ABB RAPID module: P903.mod

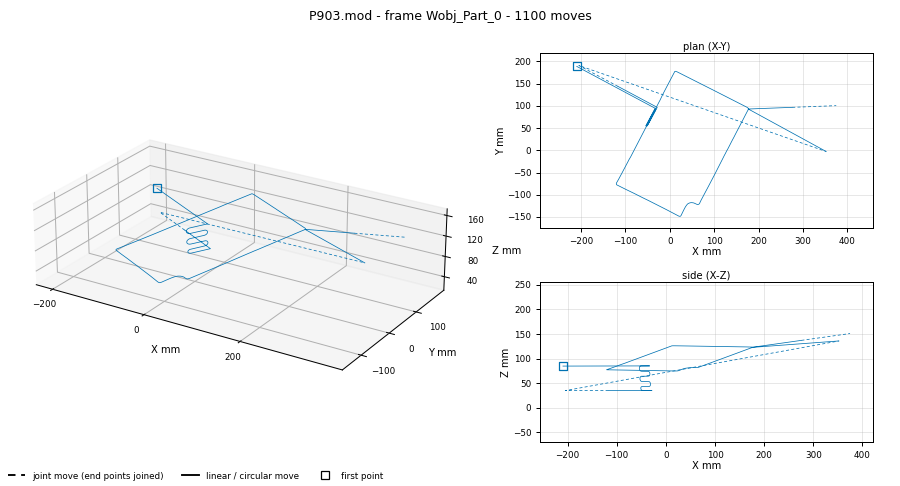
[picture p0: tool path of P903.mod in frame Wobj_Part_0, 1100 of 1110 moves have a stored position in this frame; points joined in program order, loops and branches not executed]
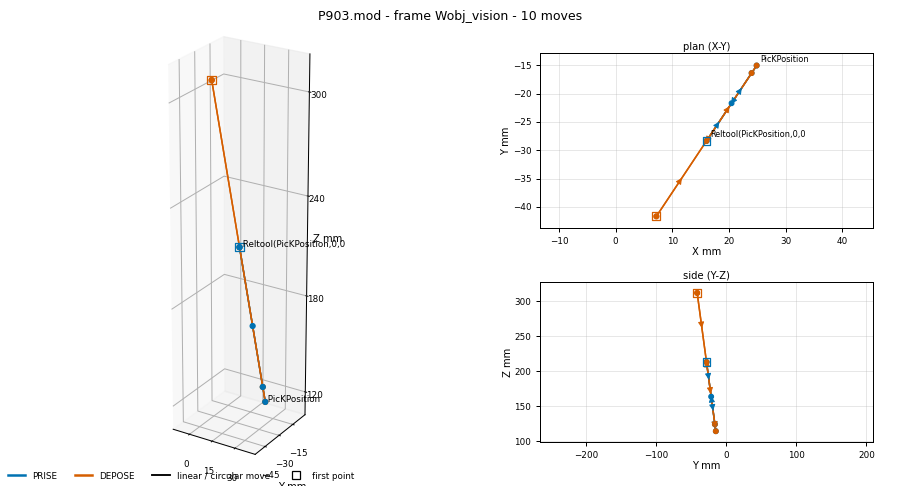
[picture p1: tool path of P903.mod in frame Wobj_vision, 10 of 1110 moves have a stored position in this frame; points joined in program order, loops and branches not executed]
MODULE P903

    ! Nom         :P903
    ! Description :
    ! Créé le     :01/06/2023 15:01:56

    LOCAL CONST SPEEDDATA VitesseLente :=[10,500,0,0];
	LOCAL CONST SPEEDDATA VitesseRapide :=[30,500,0,0];
	LOCAL CONST SPEEDDATA VitesseTronconnage :=[2,500,0,0];
	LOCAL CONST SPEEDDATA VitesseTronconnageApp :=[10,500,0,0];
    !
    !Point de prise
    LOCAL PERS Robtarget PicKPosition := [[24.8984358330106,-15.047813549993,114.680940912607],[0.072391542701378,-0.511697076202154,0.855414280882458,0.0345249882523983],[0,0,0,0],[8.999999E+09,8.999999E+09,8.999999E+09,8.999999E+09,8.999999E+09,8.999999E+09]];
	LOCAL PERS Pose Ref := [[0,0,0],[1,0,0,0]];
    !
    !Declaration des points de meulage

    !Tr_meulage_motif_1 : Meulage d'un motif
    LOCAL CONST Robtarget Tr_meulage_motif_1_0 := [[-32.91730859375,94.6825546875,85.178703125],[0.363951430919515,-0.363241574410581,0.605870778174484,-0.607054787235555],[0,0,0,0],[8.999999E+09,8.999999E+09,8.999999E+09,8.999999E+09,8.999999E+09,8.999999E+09]];
    LOCAL CONST Robtarget Tr_meulage_motif_1_1 := [[-33.3889453125,93.8007578125,85.178671875],[0.363951430919515,-0.363241574410581,0.605870778174484,-0.607054787235555],[0,0,0,0],[8.999999E+09,8.999999E+09,8.999999E+09,8.999999E+09,8.999999E+09,8.999999E+09]];
    LOCAL CONST Robtarget Tr_meulage_motif_1_2 := [[-33.8605859375,92.91896875,85.1786484375],[0.363951430919515,-0.363241574410581,0.605870778174484,-0.607054787235555],[0,0,0,0],[8.999999E+09,8.999999E+09,8.999999E+09,8.999999E+09,8.999999E+09,8.999999E+09]];
    LOCAL CONST Robtarget Tr_meulage_motif_1_3 := [[-34.33222265625,92.037171875,85.178625],[0.363951430919515,-0.363241574410581,0.605870778174484,-0.607054787235555],[0,0,0,0],[8.999999E+09,8.999999E+09,8.999999E+09,8.999999E+09,8.999999E+09,8.999999E+09]];
    LOCAL CONST Robtarget Tr_meulage_motif_1_4 := [[-34.803859375,91.1553828125,85.1786015625],[0.363951430919515,-0.363241574410581,0.605870778174484,-0.607054787235555],[0,0,0,0],[8.999999E+09,8.999999E+09,8.999999E+09,8.999999E+09,8.999999E+09,8.999999E+09]];
    LOCAL CONST Robtarget Tr_meulage_motif_1_5 := [[-35.27549609375,90.2735859375,85.178578125],[0.363951430919515,-0.363241574410581,0.605870778174484,-0.607054787235555],[0,0,0,0],[8.999999E+09,8.999999E+09,8.999999E+09,8.999999E+09,8.999999E+09,8.999999E+09]];
    LOCAL CONST Robtarget Tr_meulage_motif_1_6 := [[-35.74713671875,89.391796875,85.178546875],[0.363951430919515,-0.363241574410581,0.605870778174484,-0.607054787235555],[0,0,0,0],[8.999999E+09,8.999999E+09,8.999999E+09,8.999999E+09,8.999999E+09,8.999999E+09]];
    LOCAL CONST Robtarget Tr_meulage_motif_1_7 := [[-36.2187734375,88.5100078125,85.1785234375],[0.363951430919515,-0.363241574410581,0.605870778174484,-0.607054787235555],[0,0,0,0],[8.999999E+09,8.999999E+09,8.999999E+09,8.999999E+09,8.999999E+09,8.999999E+09]];
    LOCAL CONST Robtarget Tr_meulage_motif_1_8 := [[-36.69041015625,87.6282109375,85.1785],[0.363951430919515,-0.363241574410581,0.605870778174484,-0.607054787235555],[0,0,0,0],[8.999999E+09,8.999999E+09,8.999999E+09,8.999999E+09,8.999999E+09,8.999999E+09]];
    LOCAL CONST Robtarget Tr_meulage_motif_1_9 := [[-37.162046875,86.746421875,85.1784765625],[0.363951430919515,-0.363241574410581,0.605870778174484,-0.607054787235555],[0,0,0,0],[8.999999E+09,8.999999E+09,8.999999E+09,8.999999E+09,8.999999E+09,8.999999E+09]];
    LOCAL CONST Robtarget Tr_meulage_motif_1_10 := [[-37.6336875,85.864625,85.1784453125],[0.363951430919515,-0.363241574410581,0.605870778174484,-0.607054787235555],[0,0,0,0],[8.999999E+09,8.999999E+09,8.999999E+09,8.999999E+09,8.999999E+09,8.999999E+09]];
    LOCAL CONST Robtarget Tr_meulage_motif_1_11 := [[-38.10532421875,84.9828359375,85.178421875],[0.363951430919515,-0.363241574410581,0.605870778174484,-0.607054787235555],[0,0,0,0],[8.999999E+09,8.999999E+09,8.999999E+09,8.999999E+09,8.999999E+09,8.999999E+09]];
    LOCAL CONST Robtarget Tr_meulage_motif_1_12 := [[-38.5769609375,84.1010390625,85.1783984375],[0.363951430919515,-0.363241574410581,0.605870778174484,-0.607054787235555],[0,0,0,0],[8.999999E+09,8.999999E+09,8.999999E+09,8.999999E+09,8.999999E+09,8.999999E+09]];
    LOCAL CONST Robtarget Tr_meulage_motif_1_13 := [[-39.04859765625,83.21925,85.178375],[0.363951430919515,-0.363241574410581,0.605870778174484,-0.607054787235555],[0,0,0,0],[8.999999E+09,8.999999E+09,8.999999E+09,8.999999E+09,8.999999E+09,8.999999E+09]];
    LOCAL CONST Robtarget Tr_meulage_motif_1_14 := [[-39.52023828125,82.3374609375,85.1783515625],[0.363951430919515,-0.363241574410581,0.605870778174484,-0.607054787235555],[0,0,0,0],[8.999999E+09,8.999999E+09,8.999999E+09,8.999999E+09,8.999999E+09,8.999999E+09]];
    LOCAL CONST Robtarget Tr_meulage_motif_1_15 := [[-39.991875,81.4556640625,85.1783203125],[0.363951430919515,-0.363241574410581,0.605870778174484,-0.607054787235555],[0,0,0,0],[8.999999E+09,8.999999E+09,8.999999E+09,8.999999E+09,8.999999E+09,8.999999E+09]];
    LOCAL CONST Robtarget Tr_meulage_motif_1_16 := [[-40.46351171875,80.573875,85.178296875],[0.363951430919515,-0.363241574410581,0.605870778174484,-0.607054787235555],[0,0,0,0],[8.999999E+09,8.999999E+09,8.999999E+09,8.999999E+09,8.999999E+09,8.999999E+09]];
    LOCAL CONST Robtarget Tr_meulage_motif_1_17 := [[-40.9351484375,79.692078125,85.1782734375],[0.363951430919515,-0.363241574410581,0.605870778174484,-0.607054787235555],[0,0,0,0],[8.999999E+09,8.999999E+09,8.999999E+09,8.999999E+09,8.999999E+09,8.999999E+09]];
    LOCAL CONST Robtarget Tr_meulage_motif_1_18 := [[-41.4067890625,78.8102890625,85.17825],[0.363951430919515,-0.363241574410581,0.605870778174484,-0.607054787235555],[0,0,0,0],[8.999999E+09,8.999999E+09,8.999999E+09,8.999999E+09,8.999999E+09,8.999999E+09]];
    LOCAL CONST Robtarget Tr_meulage_motif_1_19 := [[-41.87842578125,77.9284921875,85.1782265625],[0.363951430919515,-0.363241574410581,0.605870778174484,-0.607054787235555],[0,0,0,0],[8.999999E+09,8.999999E+09,8.999999E+09,8.999999E+09,8.999999E+09,8.999999E+09]];
    LOCAL CONST Robtarget Tr_meulage_motif_1_20 := [[-42.3500625,77.046703125,85.1781953125],[0.363951430919515,-0.363241574410581,0.605870778174484,-0.607054787235555],[0,0,0,0],[8.999999E+09,8.999999E+09,8.999999E+09,8.999999E+09,8.999999E+09,8.999999E+09]];
    LOCAL CONST Robtarget Tr_meulage_motif_1_21 := [[-42.82169921875,76.1649140625,85.178171875],[0.363951430919515,-0.363241574410581,0.605870778174484,-0.607054787235555],[0,0,0,0],[8.999999E+09,8.999999E+09,8.999999E+09,8.999999E+09,8.999999E+09,8.999999E+09]];
    LOCAL CONST Robtarget Tr_meulage_motif_1_22 := [[-43.29333984375,75.2831171875,85.1781484375],[0.363951430919515,-0.363241574410581,0.605870778174484,-0.607054787235555],[0,0,0,0],[8.999999E+09,8.999999E+09,8.999999E+09,8.999999E+09,8.999999E+09,8.999999E+09]];
    LOCAL CONST Robtarget Tr_meulage_motif_1_23 := [[-43.7649765625,74.401328125,85.178125],[0.363951430919515,-0.363241574410581,0.605870778174484,-0.607054787235555],[0,0,0,0],[8.999999E+09,8.999999E+09,8.999999E+09,8.999999E+09,8.999999E+09,8.999999E+09]];
    LOCAL CONST Robtarget Tr_meulage_motif_1_24 := [[-44.23661328125,73.51953125,85.17809375],[0.363951430919515,-0.363241574410581,0.605870778174484,-0.607054787235555],[0,0,0,0],[8.999999E+09,8.999999E+09,8.999999E+09,8.999999E+09,8.999999E+09,8.999999E+09]];
    LOCAL CONST Robtarget Tr_meulage_motif_1_25 := [[-44.70825,72.6377421875,85.1780703125],[0.363951430919515,-0.363241574410581,0.605870778174484,-0.607054787235555],[0,0,0,0],[8.999999E+09,8.999999E+09,8.999999E+09,8.999999E+09,8.999999E+09,8.999999E+09]];
    LOCAL CONST Robtarget Tr_meulage_motif_1_26 := [[-45.179890625,71.7559453125,85.178046875],[0.363951430919515,-0.363241574410581,0.605870778174484,-0.607054787235555],[0,0,0,0],[8.999999E+09,8.999999E+09,8.999999E+09,8.999999E+09,8.999999E+09,8.999999E+09]];
    LOCAL CONST Robtarget Tr_meulage_motif_1_27 := [[-45.65152734375,70.87415625,85.1780234375],[0.363951430919515,-0.363241574410581,0.605870778174484,-0.607054787235555],[0,0,0,0],[8.999999E+09,8.999999E+09,8.999999E+09,8.999999E+09,8.999999E+09,8.999999E+09]];
    LOCAL CONST Robtarget Tr_meulage_motif_1_28 := [[-46.1231640625,69.9923671875,85.178],[0.363951430919515,-0.363241574410581,0.605870778174484,-0.607054787235555],[0,0,0,0],[8.999999E+09,8.999999E+09,8.999999E+09,8.999999E+09,8.999999E+09,8.999999E+09]];
    LOCAL CONST Robtarget Tr_meulage_motif_1_29 := [[-46.59480078125,69.1105703125,85.17796875],[0.363951430919515,-0.363241574410581,0.605870778174484,-0.607054787235555],[0,0,0,0],[8.999999E+09,8.999999E+09,8.999999E+09,8.999999E+09,8.999999E+09,8.999999E+09]];
    LOCAL CONST Robtarget Tr_meulage_motif_1_30 := [[-47.06644140625,68.22878125,85.1779453125],[0.363951430919515,-0.363241574410581,0.605870778174484,-0.607054787235555],[0,0,0,0],[8.999999E+09,8.999999E+09,8.999999E+09,8.999999E+09,8.999999E+09,8.999999E+09]];
    LOCAL CONST Robtarget Tr_meulage_motif_1_31 := [[-47.538078125,67.346984375,85.177921875],[0.363951430919515,-0.363241574410581,0.605870778174484,-0.607054787235555],[0,0,0,0],[8.999999E+09,8.999999E+09,8.999999E+09,8.999999E+09,8.999999E+09,8.999999E+09]];
    LOCAL CONST Robtarget Tr_meulage_motif_1_32 := [[-48.00971484375,66.4651953125,85.1778984375],[0.363951430919515,-0.363241574410581,0.605870778174484,-0.607054787235555],[0,0,0,0],[8.999999E+09,8.999999E+09,8.999999E+09,8.999999E+09,8.999999E+09,8.999999E+09]];
    LOCAL CONST Robtarget Tr_meulage_motif_1_33 := [[-48.4813515625,65.5833984375,85.1778671875],[0.363951430919515,-0.363241574410581,0.605870778174484,-0.607054787235555],[0,0,0,0],[8.999999E+09,8.999999E+09,8.999999E+09,8.999999E+09,8.999999E+09,8.999999E+09]];
    LOCAL CONST Robtarget Tr_meulage_motif_1_34 := [[-48.9529921875,64.701609375,85.17784375],[0.363951430919515,-0.363241574410581,0.605870778174484,-0.607054787235555],[0,0,0,0],[8.999999E+09,8.999999E+09,8.999999E+09,8.999999E+09,8.999999E+09,8.999999E+09]];
    LOCAL CONST Robtarget Tr_meulage_motif_1_35 := [[-49.42462890625,63.81981640625,85.1778203125],[0.363951430919515,-0.363241574410581,0.605870778174484,-0.607054787235555],[0,0,0,0],[8.999999E+09,8.999999E+09,8.999999E+09,8.999999E+09,8.999999E+09,8.999999E+09]];
    LOCAL CONST Robtarget Tr_meulage_motif_1_36 := [[-49.896265625,62.9380234375,85.177796875],[0.363951430919515,-0.363241574410581,0.605870778174484,-0.607054787235555],[0,0,0,0],[8.999999E+09,8.999999E+09,8.999999E+09,8.999999E+09,8.999999E+09,8.999999E+09]];
    LOCAL CONST Robtarget Tr_meulage_motif_1_37 := [[-50.36790234375,62.05623046875,85.1777734375],[0.363951430919515,-0.363241574410581,0.605870778174484,-0.607054787235555],[0,0,0,0],[8.999999E+09,8.999999E+09,8.999999E+09,8.999999E+09,8.999999E+09,8.999999E+09]];
    LOCAL CONST Robtarget Tr_meulage_motif_1_38 := [[-50.83954296875,61.1744375,85.1777421875],[0.363951430919515,-0.363241574410581,0.605870778174484,-0.607054787235555],[0,0,0,0],[8.999999E+09,8.999999E+09,8.999999E+09,8.999999E+09,8.999999E+09,8.999999E+09]];
    LOCAL CONST Robtarget Tr_meulage_motif_1_39 := [[-51.3013984375,60.2958515625,85.067359375],[0.363951430919515,-0.363241574410581,0.605870778174484,-0.607054787235555],[0,0,0,0],[8.999999E+09,8.999999E+09,8.999999E+09,8.999999E+09,8.999999E+09,8.999999E+09]];
    LOCAL CONST Robtarget Tr_meulage_motif_1_40 := [[-51.7358203125,59.45483203125,84.856578125],[0.363951430919515,-0.363241574410581,0.605870778174484,-0.607054787235555],[0,0,0,0],[8.999999E+09,8.999999E+09,8.999999E+09,8.999999E+09,8.999999E+09,8.999999E+09]];
    LOCAL CONST Robtarget Tr_meulage_motif_1_41 := [[-52.12257421875,58.694671875,84.58528125],[0.363951430919515,-0.363241574410581,0.605870778174484,-0.607054787235555],[0,0,0,0],[8.999999E+09,8.999999E+09,8.999999E+09,8.999999E+09,8.999999E+09,8.999999E+09]];
    LOCAL CONST Robtarget Tr_meulage_motif_1_42 := [[-52.4606171875,58.025015625,84.3098984375],[0.363951430919515,-0.363241574410581,0.605870778174484,-0.607054787235555],[0,0,0,0],[8.999999E+09,8.999999E+09,8.999999E+09,8.999999E+09,8.999999E+09,8.999999E+09]];
    LOCAL CONST Robtarget Tr_meulage_motif_1_43 := [[-52.94496484375,57.0354296875,83.695015625],[0.363951430919515,-0.363241574410581,0.605870778174484,-0.607054787235555],[0,0,0,0],[8.999999E+09,8.999999E+09,8.999999E+09,8.999999E+09,8.999999E+09,8.999999E+09]];
    LOCAL CONST Robtarget Tr_meulage_motif_1_44 := [[-53.37976953125,56.10688671875,82.84909375],[0.363951430919515,-0.363241574410581,0.605870778174484,-0.607054787235555],[0,0,0,0],[8.999999E+09,8.999999E+09,8.999999E+09,8.999999E+09,8.999999E+09,8.999999E+09]];
    LOCAL CONST Robtarget Tr_meulage_motif_1_45 := [[-53.72146875,55.328390625,81.8273125],[0.363951430919515,-0.363241574410581,0.605870778174484,-0.607054787235555],[0,0,0,0],[8.999999E+09,8.999999E+09,8.999999E+09,8.999999E+09,8.999999E+09,8.999999E+09]];
    LOCAL CONST Robtarget Tr_meulage_motif_1_46 := [[-53.888375,54.86409765625,80.7134296875],[0.363951430919515,-0.363241574410581,0.605870778174484,-0.607054787235555],[0,0,0,0],[8.999999E+09,8.999999E+09,8.999999E+09,8.999999E+09,8.999999E+09,8.999999E+09]];
    LOCAL CONST Robtarget Tr_meulage_motif_1_47 := [[-53.86165625,54.81913671875,80.0188984375],[0.363951430919515,-0.363241574410581,0.605870778174484,-0.607054787235555],[0,0,0,0],[8.999999E+09,8.999999E+09,8.999999E+09,8.999999E+09,8.999999E+09,8.999999E+09]];
    LOCAL CONST Robtarget Tr_meulage_motif_1_48 := [[-53.824140625,54.79908984375,79.359015625],[0.363951430919515,-0.363241574410581,0.605870778174484,-0.607054787235555],[0,0,0,0],[8.999999E+09,8.999999E+09,8.999999E+09,8.999999E+09,8.999999E+09,8.999999E+09]];
    LOCAL CONST Robtarget Tr_meulage_motif_1_49 := [[-53.76075390625,54.82743359375,78.699296875],[0.363951430919515,-0.363241574410581,0.605870778174484,-0.607054787235555],[0,0,0,0],[8.999999E+09,8.999999E+09,8.999999E+09,8.999999E+09,8.999999E+09,8.999999E+09]];
    LOCAL CONST Robtarget Tr_meulage_motif_1_50 := [[-53.463265625,55.233359375,77.59984375],[0.363951430919515,-0.363241574410581,0.605870778174484,-0.607054787235555],[0,0,0,0],[8.999999E+09,8.999999E+09,8.999999E+09,8.999999E+09,8.999999E+09,8.999999E+09]];
    LOCAL CONST Robtarget Tr_meulage_motif_1_51 := [[-53.002140625,55.95820703125,76.5953203125],[0.363951430919515,-0.363241574410581,0.605870778174484,-0.607054787235555],[0,0,0,0],[8.999999E+09,8.999999E+09,8.999999E+09,8.999999E+09,8.999999E+09,8.999999E+09]];
    LOCAL CONST Robtarget Tr_meulage_motif_1_52 := [[-52.4724375,56.83551171875,75.7681875],[0.363951430919515,-0.363241574410581,0.605870778174484,-0.607054787235555],[0,0,0,0],[8.999999E+09,8.999999E+09,8.999999E+09,8.999999E+09,8.999999E+09,8.999999E+09]];
    LOCAL CONST Robtarget Tr_meulage_motif_1_53 := [[-52.12592578125,57.42938671875,75.3732734375],[0.363951430919515,-0.363241574410581,0.605870778174484,-0.607054787235555],[0,0,0,0],[8.999999E+09,8.999999E+09,8.999999E+09,8.999999E+09,8.999999E+09,8.999999E+09]];
    LOCAL CONST Robtarget Tr_meulage_motif_1_54 := [[-51.55203515625,58.435859375,74.88678125],[0.363951430919515,-0.363241574410581,0.605870778174484,-0.607054787235555],[0,0,0,0],[8.999999E+09,8.999999E+09,8.999999E+09,8.999999E+09,8.999999E+09,8.999999E+09]];
    LOCAL CONST Robtarget Tr_meulage_motif_1_55 := [[-51.13850390625,59.17299609375,74.6232578125],[0.363951430919515,-0.363241574410581,0.605870778174484,-0.607054787235555],[0,0,0,0],[8.999999E+09,8.999999E+09,8.999999E+09,8.999999E+09,8.999999E+09,8.999999E+09]];
    LOCAL CONST Robtarget Tr_meulage_motif_1_56 := [[-50.68733984375,59.98862890625,74.419234375],[0.363951430919515,-0.363241574410581,0.605870778174484,-0.607054787235555],[0,0,0,0],[8.999999E+09,8.999999E+09,8.999999E+09,8.999999E+09,8.999999E+09,8.999999E+09]];
    LOCAL CONST Robtarget Tr_meulage_motif_1_57 := [[-50.218234375,60.85087109375,74.310890625],[0.363951430919515,-0.363241574410581,0.605870778174484,-0.607054787235555],[0,0,0,0],[8.999999E+09,8.999999E+09,8.999999E+09,8.999999E+09,8.999999E+09,8.999999E+09]];
    LOCAL CONST Robtarget Tr_meulage_motif_1_58 := [[-49.74383203125,61.72275,74.2005546875],[0.363951430919515,-0.363241574410581,0.605870778174484,-0.607054787235555],[0,0,0,0],[8.999999E+09,8.999999E+09,8.999999E+09,8.999999E+09,8.999999E+09,8.999999E+09]];
    LOCAL CONST Robtarget Tr_meulage_motif_1_59 := [[-49.2721953125,62.60454296875,74.200578125],[0.363951430919515,-0.363241574410581,0.605870778174484,-0.607054787235555],[0,0,0,0],[8.999999E+09,8.999999E+09,8.999999E+09,8.999999E+09,8.999999E+09,8.999999E+09]];
    LOCAL CONST Robtarget Tr_meulage_motif_1_60 := [[-48.8005546875,63.4863359375,74.2006015625],[0.363951430919515,-0.363241574410581,0.605870778174484,-0.607054787235555],[0,0,0,0],[8.999999E+09,8.999999E+09,8.999999E+09,8.999999E+09,8.999999E+09,8.999999E+09]];
    LOCAL CONST Robtarget Tr_meulage_motif_1_61 := [[-48.32891796875,64.36812890625,74.200625],[0.363951430919515,-0.363241574410581,0.605870778174484,-0.607054787235555],[0,0,0,0],[8.999999E+09,8.999999E+09,8.999999E+09,8.999999E+09,8.999999E+09,8.999999E+09]];
    LOCAL CONST Robtarget Tr_meulage_motif_1_62 := [[-47.85728125,65.249921875,74.20065625],[0.363951430919515,-0.363241574410581,0.605870778174484,-0.607054787235555],[0,0,0,0],[8.999999E+09,8.999999E+09,8.999999E+09,8.999999E+09,8.999999E+09,8.999999E+09]];
    LOCAL CONST Robtarget Tr_meulage_motif_1_63 := [[-47.38564453125,66.1317109375,74.2006796875],[0.363951430919515,-0.363241574410581,0.605870778174484,-0.607054787235555],[0,0,0,0],[8.999999E+09,8.999999E+09,8.999999E+09,8.999999E+09,8.999999E+09,8.999999E+09]];
    LOCAL CONST Robtarget Tr_meulage_motif_1_64 := [[-46.91400390625,67.0135078125,74.200703125],[0.363951430919515,-0.363241574410581,0.605870778174484,-0.607054787235555],[0,0,0,0],[8.999999E+09,8.999999E+09,8.999999E+09,8.999999E+09,8.999999E+09,8.999999E+09]];
    LOCAL CONST Robtarget Tr_meulage_motif_1_65 := [[-46.4423671875,67.895296875,74.2007265625],[0.363951430919515,-0.363241574410581,0.605870778174484,-0.607054787235555],[0,0,0,0],[8.999999E+09,8.999999E+09,8.999999E+09,8.999999E+09,8.999999E+09,8.999999E+09]];
    LOCAL CONST Robtarget Tr_meulage_motif_1_66 := [[-45.97073046875,68.77709375,74.20075],[0.363951430919515,-0.363241574410581,0.605870778174484,-0.607054787235555],[0,0,0,0],[8.999999E+09,8.999999E+09,8.999999E+09,8.999999E+09,8.999999E+09,8.999999E+09]];
    LOCAL CONST Robtarget Tr_meulage_motif_1_67 := [[-45.49909375,69.6588828125,74.20078125],[0.363951430919515,-0.363241574410581,0.605870778174484,-0.607054787235555],[0,0,0,0],[8.999999E+09,8.999999E+09,8.999999E+09,8.999999E+09,8.999999E+09,8.999999E+09]];
    LOCAL CONST Robtarget Tr_meulage_motif_1_68 := [[-45.027453125,70.540671875,74.2008046875],[0.363951430919515,-0.363241574410581,0.605870778174484,-0.607054787235555],[0,0,0,0],[8.999999E+09,8.999999E+09,8.999999E+09,8.999999E+09,8.999999E+09,8.999999E+09]];
    LOCAL CONST Robtarget Tr_meulage_motif_1_69 := [[-44.55581640625,71.42246875,74.200828125],[0.363951430919515,-0.363241574410581,0.605870778174484,-0.607054787235555],[0,0,0,0],[8.999999E+09,8.999999E+09,8.999999E+09,8.999999E+09,8.999999E+09,8.999999E+09]];
    LOCAL CONST Robtarget Tr_meulage_motif_1_70 := [[-44.0841796875,72.3042578125,74.2008515625],[0.363951430919515,-0.363241574410581,0.605870778174484,-0.607054787235555],[0,0,0,0],[8.999999E+09,8.999999E+09,8.999999E+09,8.999999E+09,8.999999E+09,8.999999E+09]];
    LOCAL CONST Robtarget Tr_meulage_motif_1_71 := [[-43.61254296875,73.1860546875,74.200875],[0.363951430919515,-0.363241574410581,0.605870778174484,-0.607054787235555],[0,0,0,0],[8.999999E+09,8.999999E+09,8.999999E+09,8.999999E+09,8.999999E+09,8.999999E+09]];
    LOCAL CONST Robtarget Tr_meulage_motif_1_72 := [[-43.14090234375,74.06784375,74.20090625],[0.363951430919515,-0.363241574410581,0.605870778174484,-0.607054787235555],[0,0,0,0],[8.999999E+09,8.999999E+09,8.999999E+09,8.999999E+09,8.999999E+09,8.999999E+09]];
    LOCAL CONST Robtarget Tr_meulage_motif_1_73 := [[-42.669265625,74.949640625,74.2009296875],[0.363951430919515,-0.363241574410581,0.605870778174484,-0.607054787235555],[0,0,0,0],[8.999999E+09,8.999999E+09,8.999999E+09,8.999999E+09,8.999999E+09,8.999999E+09]];
    LOCAL CONST Robtarget Tr_meulage_motif_1_74 := [[-42.19762890625,75.8314296875,74.200953125],[0.363951430919515,-0.363241574410581,0.605870778174484,-0.607054787235555],[0,0,0,0],[8.999999E+09,8.999999E+09,8.999999E+09,8.999999E+09,8.999999E+09,8.999999E+09]];
    LOCAL CONST Robtarget Tr_meulage_motif_1_75 := [[-41.7259921875,76.71321875,74.2009765625],[0.363951430919515,-0.363241574410581,0.605870778174484,-0.607054787235555],[0,0,0,0],[8.999999E+09,8.999999E+09,8.999999E+09,8.999999E+09,8.999999E+09,8.999999E+09]];
    LOCAL CONST Robtarget Tr_meulage_motif_1_76 := [[-41.2543515625,77.595015625,74.2010078125],[0.363951430919515,-0.363241574410581,0.605870778174484,-0.607054787235555],[0,0,0,0],[8.999999E+09,8.999999E+09,8.999999E+09,8.999999E+09,8.999999E+09,8.999999E+09]];
    LOCAL CONST Robtarget Tr_meulage_motif_1_77 := [[-40.78271484375,78.4768046875,74.20103125],[0.363951430919515,-0.363241574410581,0.605870778174484,-0.607054787235555],[0,0,0,0],[8.999999E+09,8.999999E+09,8.999999E+09,8.999999E+09,8.999999E+09,8.999999E+09]];
    LOCAL CONST Robtarget Tr_meulage_motif_1_78 := [[-40.311078125,79.3586015625,74.2010546875],[0.363951430919515,-0.363241574410581,0.605870778174484,-0.607054787235555],[0,0,0,0],[8.999999E+09,8.999999E+09,8.999999E+09,8.999999E+09,8.999999E+09,8.999999E+09]];
    LOCAL CONST Robtarget Tr_meulage_motif_1_79 := [[-39.83944140625,80.240390625,74.201078125],[0.363951430919515,-0.363241574410581,0.605870778174484,-0.607054787235555],[0,0,0,0],[8.999999E+09,8.999999E+09,8.999999E+09,8.999999E+09,8.999999E+09,8.999999E+09]];
    LOCAL CONST Robtarget Tr_meulage_motif_1_80 := [[-39.36780078125,81.1221875,74.2011015625],[0.363951430919515,-0.363241574410581,0.605870778174484,-0.607054787235555],[0,0,0,0],[8.999999E+09,8.999999E+09,8.999999E+09,8.999999E+09,8.999999E+09,8.999999E+09]];
    LOCAL CONST Robtarget Tr_meulage_motif_1_81 := [[-38.8961640625,82.0039765625,74.2011328125],[0.363951430919515,-0.363241574410581,0.605870778174484,-0.607054787235555],[0,0,0,0],[8.999999E+09,8.999999E+09,8.999999E+09,8.999999E+09,8.999999E+09,8.999999E+09]];
    LOCAL CONST Robtarget Tr_meulage_motif_1_82 := [[-38.42452734375,82.8857734375,74.20115625],[0.363951430919515,-0.363241574410581,0.605870778174484,-0.607054787235555],[0,0,0,0],[8.999999E+09,8.999999E+09,8.999999E+09,8.999999E+09,8.999999E+09,8.999999E+09]];
    LOCAL CONST Robtarget Tr_meulage_motif_1_83 := [[-37.952890625,83.7675625,74.2011796875],[0.363951430919515,-0.363241574410581,0.605870778174484,-0.607054787235555],[0,0,0,0],[8.999999E+09,8.999999E+09,8.999999E+09,8.999999E+09,8.999999E+09,8.999999E+09]];
    LOCAL CONST Robtarget Tr_meulage_motif_1_84 := [[-37.48125,84.6493515625,74.201203125],[0.363951430919515,-0.363241574410581,0.605870778174484,-0.607054787235555],[0,0,0,0],[8.999999E+09,8.999999E+09,8.999999E+09,8.999999E+09,8.999999E+09,8.999999E+09]];
    LOCAL CONST Robtarget Tr_meulage_motif_1_85 := [[-37.00961328125,85.5311484375,74.2012265625],[0.363951430919515,-0.363241574410581,0.605870778174484,-0.607054787235555],[0,0,0,0],[8.999999E+09,8.999999E+09,8.999999E+09,8.999999E+09,8.999999E+09,8.999999E+09]];
    LOCAL CONST Robtarget Tr_meulage_motif_1_86 := [[-36.5379765625,86.4129375,74.2012578125],[0.363951430919515,-0.363241574410581,0.605870778174484,-0.607054787235555],[0,0,0,0],[8.999999E+09,8.999999E+09,8.999999E+09,8.999999E+09,8.999999E+09,8.999999E+09]];
    LOCAL CONST Robtarget Tr_meulage_motif_1_87 := [[-36.06633984375,87.294734375,74.20128125],[0.363951430919515,-0.363241574410581,0.605870778174484,-0.607054787235555],[0,0,0,0],[8.999999E+09,8.999999E+09,8.999999E+09,8.999999E+09,8.999999E+09,8.999999E+09]];
    LOCAL CONST Robtarget Tr_meulage_motif_1_88 := [[-35.59469921875,88.1765234375,74.2013046875],[0.363951430919515,-0.363241574410581,0.605870778174484,-0.607054787235555],[0,0,0,0],[8.999999E+09,8.999999E+09,8.999999E+09,8.999999E+09,8.999999E+09,8.999999E+09]];
    LOCAL CONST Robtarget Tr_meulage_motif_1_89 := [[-35.120296875,89.04840625,74.09096875],[0.363951430919515,-0.363241574410581,0.605870778174484,-0.607054787235555],[0,0,0,0],[8.999999E+09,8.999999E+09,8.999999E+09,8.999999E+09,8.999999E+09,8.999999E+09]];
    LOCAL CONST Robtarget Tr_meulage_motif_1_90 := [[-34.66191015625,89.8766171875,73.8802421875],[0.363951430919515,-0.363241574410581,0.605870778174484,-0.607054787235555],[0,0,0,0],[8.999999E+09,8.999999E+09,8.999999E+09,8.999999E+09,8.999999E+09,8.999999E+09]];
    LOCAL CONST Robtarget Tr_meulage_motif_1_91 := [[-34.2443125,90.620296875,73.6089765625],[0.363951430919515,-0.363241574410581,0.605870778174484,-0.607054787235555],[0,0,0,0],[8.999999E+09,8.999999E+09,8.999999E+09,8.999999E+09,8.999999E+09,8.999999E+09]];
    LOCAL CONST Robtarget Tr_meulage_motif_1_92 := [[-33.89148828125,91.2384765625,73.30546875],[0.363951430919515,-0.363241574410581,0.605870778174484,-0.607054787235555],[0,0,0,0],[8.999999E+09,8.999999E+09,8.999999E+09,8.999999E+09,8.999999E+09,8.999999E+09]];
    LOCAL CONST Robtarget Tr_meulage_motif_1_93 := [[-33.36600390625,92.130578125,72.6443359375],[0.363951430919515,-0.363241574410581,0.605870778174484,-0.607054787235555],[0,0,0,0],[8.999999E+09,8.999999E+09,8.999999E+09,8.999999E+09,8.999999E+09,8.999999E+09]];
    LOCAL CONST Robtarget Tr_meulage_motif_1_94 := [[-32.8894453125,92.8985546875,71.7442890625],[0.363951430919515,-0.363241574410581,0.605870778174484,-0.607054787235555],[0,0,0,0],[8.999999E+09,8.999999E+09,8.999999E+09,8.999999E+09,8.999999E+09,8.999999E+09]];
    LOCAL CONST Robtarget Tr_meulage_motif_1_95 := [[-32.5777890625,93.3385703125,70.7004375],[0.363951430919515,-0.363241574410581,0.605870778174484,-0.607054787235555],[0,0,0,0],[8.999999E+09,8.999999E+09,8.999999E+09,8.999999E+09,8.999999E+09,8.999999E+09]];
    LOCAL CONST Robtarget Tr_meulage_motif_1_96 := [[-32.451310546875,93.4804921875,70.0086640625],[0.363951430919515,-0.363241574410581,0.605870778174484,-0.607054787235555],[0,0,0,0],[8.999999E+09,8.999999E+09,8.999999E+09,8.999999E+09,8.999999E+09,8.999999E+09]];
    LOCAL CONST Robtarget Tr_meulage_motif_1_97 := [[-32.377513671875,93.5134453125,69.2402578125],[0.363951430919515,-0.363241574410581,0.605870778174484,-0.607054787235555],[0,0,0,0],[8.999999E+09,8.999999E+09,8.999999E+09,8.999999E+09,8.999999E+09,8.999999E+09]];
    LOCAL CONST Robtarget Tr_meulage_motif_1_98 := [[-32.36540625,93.4310859375,68.4719765625],[0.363951430919515,-0.363241574410581,0.605870778174484,-0.607054787235555],[0,0,0,0],[8.999999E+09,8.999999E+09,8.999999E+09,8.999999E+09,8.999999E+09,8.999999E+09]];
    LOCAL CONST Robtarget Tr_meulage_motif_1_99 := [[-32.500427734375,93.0274921875,67.3660078125],[0.363951430919515,-0.363241574410581,0.605870778174484,-0.607054787235555],[0,0,0,0],[8.999999E+09,8.999999E+09,8.999999E+09,8.999999E+09,8.999999E+09,8.999999E+09]];
    LOCAL CONST Robtarget Tr_meulage_motif_1_100 := [[-32.66260546875,92.6443984375,66.7815234375],[0.363951430919515,-0.363241574410581,0.605870778174484,-0.607054787235555],[0,0,0,0],[8.999999E+09,8.999999E+09,8.999999E+09,8.999999E+09,8.999999E+09,8.999999E+09]];
    LOCAL CONST Robtarget Tr_meulage_motif_1_101 := [[-33.03067578125,91.8352421875,65.89621875],[0.363951430919515,-0.363241574410581,0.605870778174484,-0.607054787235555],[0,0,0,0],[8.999999E+09,8.999999E+09,8.999999E+09,8.999999E+09,8.999999E+09,8.999999E+09]];
    LOCAL CONST Robtarget Tr_meulage_motif_1_102 := [[-33.28340234375,91.3062265625,65.48274609375],[0.363951430919515,-0.363241574410581,0.605870778174484,-0.607054787235555],[0,0,0,0],[8.999999E+09,8.999999E+09,8.999999E+09,8.999999E+09,8.999999E+09,8.999999E+09]];
    LOCAL CONST Robtarget Tr_meulage_motif_1_103 := [[-33.77978125,90.30396875,64.93975],[0.363951430919515,-0.363241574410581,0.605870778174484,-0.607054787235555],[0,0,0,0],[8.999999E+09,8.999999E+09,8.999999E+09,8.999999E+09,8.999999E+09,8.999999E+09]];
    LOCAL CONST Robtarget Tr_meulage_motif_1_104 := [[-34.1523984375,89.5670078125,64.64484375],[0.363951430919515,-0.363241574410581,0.605870778174484,-0.607054787235555],[0,0,0,0],[8.999999E+09,8.999999E+09,8.999999E+09,8.999999E+09,8.999999E+09,8.999999E+09]];
    LOCAL CONST Robtarget Tr_meulage_motif_1_105 := [[-34.58036328125,88.738984375,64.4407734375],[0.363951430919515,-0.363241574410581,0.605870778174484,-0.607054787235555],[0,0,0,0],[8.999999E+09,8.999999E+09,8.999999E+09,8.999999E+09,8.999999E+09,8.999999E+09]];
    LOCAL CONST Robtarget Tr_meulage_motif_1_106 := [[-35.03714453125,87.87015625,64.3323828125],[0.363951430919515,-0.363241574410581,0.605870778174484,-0.607054787235555],[0,0,0,0],[8.999999E+09,8.999999E+09,8.999999E+09,8.999999E+09,8.999999E+09,8.999999E+09]];
    LOCAL CONST Robtarget Tr_meulage_motif_1_107 := [[-35.499,86.9915703125,64.2219921875],[0.363951430919515,-0.363241574410581,0.605870778174484,-0.607054787235555],[0,0,0,0],[8.999999E+09,8.999999E+09,8.999999E+09,8.999999E+09,8.999999E+09,8.999999E+09]];
    LOCAL CONST Robtarget Tr_meulage_motif_1_108 := [[-35.97063671875,86.1097734375,64.22196484375],[0.363951430919515,-0.363241574410581,0.605870778174484,-0.607054787235555],[0,0,0,0],[8.999999E+09,8.999999E+09,8.999999E+09,8.999999E+09,8.999999E+09,8.999999E+09]];
    LOCAL CONST Robtarget Tr_meulage_motif_1_109 := [[-36.4422734375,85.227984375,64.22194140625],[0.363951430919515,-0.363241574410581,0.605870778174484,-0.607054787235555],[0,0,0,0],[8.999999E+09,8.999999E+09,8.999999E+09,8.999999E+09,8.999999E+09,8.999999E+09]];
    LOCAL CONST Robtarget Tr_meulage_motif_1_110 := [[-36.9139140625,84.3461875,64.2219140625],[0.363951430919515,-0.363241574410581,0.605870778174484,-0.607054787235555],[0,0,0,0],[8.999999E+09,8.999999E+09,8.999999E+09,8.999999E+09,8.999999E+09,8.999999E+09]];
    LOCAL CONST Robtarget Tr_meulage_motif_1_111 := [[-37.38555078125,83.4643984375,64.221890625],[0.363951430919515,-0.363241574410581,0.605870778174484,-0.607054787235555],[0,0,0,0],[8.999999E+09,8.999999E+09,8.999999E+09,8.999999E+09,8.999999E+09,8.999999E+09]];
    LOCAL CONST Robtarget Tr_meulage_motif_1_112 := [[-37.8571875,82.582609375,64.2218671875],[0.363951430919515,-0.363241574410581,0.605870778174484,-0.607054787235555],[0,0,0,0],[8.999999E+09,8.999999E+09,8.999999E+09,8.999999E+09,8.999999E+09,8.999999E+09]];
    LOCAL CONST Robtarget Tr_meulage_motif_1_113 := [[-38.32882421875,81.7008125,64.22183984375],[0.363951430919515,-0.363241574410581,0.605870778174484,-0.607054787235555],[0,0,0,0],[8.999999E+09,8.999999E+09,8.999999E+09,8.999999E+09,8.999999E+09,8.999999E+09]];
    LOCAL CONST Robtarget Tr_meulage_motif_1_114 := [[-38.80046484375,80.8190234375,64.22181640625],[0.363951430919515,-0.363241574410581,0.605870778174484,-0.607054787235555],[0,0,0,0],[8.999999E+09,8.999999E+09,8.999999E+09,8.999999E+09,8.999999E+09,8.999999E+09]];
    LOCAL CONST Robtarget Tr_meulage_motif_1_115 := [[-39.2721015625,79.9372265625,64.2217890625],[0.363951430919515,-0.363241574410581,0.605870778174484,-0.607054787235555],[0,0,0,0],[8.999999E+09,8.999999E+09,8.999999E+09,8.999999E+09,8.999999E+09,8.999999E+09]];
    LOCAL CONST Robtarget Tr_meulage_motif_1_116 := [[-39.74373828125,79.0554375,64.221765625],[0.363951430919515,-0.363241574410581,0.605870778174484,-0.607054787235555],[0,0,0,0],[8.999999E+09,8.999999E+09,8.999999E+09,8.999999E+09,8.999999E+09,8.999999E+09]];
    LOCAL CONST Robtarget Tr_meulage_motif_1_117 := [[-40.215375,78.173640625,64.22173828125],[0.363951430919515,-0.363241574410581,0.605870778174484,-0.607054787235555],[0,0,0,0],[8.999999E+09,8.999999E+09,8.999999E+09,8.999999E+09,8.999999E+09,8.999999E+09]];
    LOCAL CONST Robtarget Tr_meulage_motif_1_118 := [[-40.687015625,77.2918515625,64.22171484375],[0.363951430919515,-0.363241574410581,0.605870778174484,-0.607054787235555],[0,0,0,0],[8.999999E+09,8.999999E+09,8.999999E+09,8.999999E+09,8.999999E+09,8.999999E+09]];
    LOCAL CONST Robtarget Tr_meulage_motif_1_119 := [[-41.15865234375,76.4100625,64.22169140625],[0.363951430919515,-0.363241574410581,0.605870778174484,-0.607054787235555],[0,0,0,0],[8.999999E+09,8.999999E+09,8.999999E+09,8.999999E+09,8.999999E+09,8.999999E+09]];
    LOCAL CONST Robtarget Tr_meulage_motif_1_120 := [[-41.6302890625,75.528265625,64.2216640625],[0.363951430919515,-0.363241574410581,0.605870778174484,-0.607054787235555],[0,0,0,0],[8.999999E+09,8.999999E+09,8.999999E+09,8.999999E+09,8.999999E+09,8.999999E+09]];
    LOCAL CONST Robtarget Tr_meulage_motif_1_121 := [[-42.10192578125,74.6464765625,64.221640625],[0.363951430919515,-0.363241574410581,0.605870778174484,-0.607054787235555],[0,0,0,0],[8.999999E+09,8.999999E+09,8.999999E+09,8.999999E+09,8.999999E+09,8.999999E+09]];
    LOCAL CONST Robtarget Tr_meulage_motif_1_122 := [[-42.57356640625,73.7646796875,64.22161328125],[0.363951430919515,-0.363241574410581,0.605870778174484,-0.607054787235555],[0,0,0,0],[8.999999E+09,8.999999E+09,8.999999E+09,8.999999E+09,8.999999E+09,8.999999E+09]];
    LOCAL CONST Robtarget Tr_meulage_motif_1_123 := [[-43.045203125,72.882890625,64.22158984375],[0.363951430919515,-0.363241574410581,0.605870778174484,-0.607054787235555],[0,0,0,0],[8.999999E+09,8.999999E+09,8.999999E+09,8.999999E+09,8.999999E+09,8.999999E+09]];
    LOCAL CONST Robtarget Tr_meulage_motif_1_124 := [[-43.51683984375,72.00109375,64.2215625],[0.363951430919515,-0.363241574410581,0.605870778174484,-0.607054787235555],[0,0,0,0],[8.999999E+09,8.999999E+09,8.999999E+09,8.999999E+09,8.999999E+09,8.999999E+09]];
    LOCAL CONST Robtarget Tr_meulage_motif_1_125 := [[-43.9884765625,71.1193046875,64.2215390625],[0.363951430919515,-0.363241574410581,0.605870778174484,-0.607054787235555],[0,0,0,0],[8.999999E+09,8.999999E+09,8.999999E+09,8.999999E+09,8.999999E+09,8.999999E+09]];
    LOCAL CONST Robtarget Tr_meulage_motif_1_126 := [[-44.4601171875,70.237515625,64.221515625],[0.363951430919515,-0.363241574410581,0.605870778174484,-0.607054787235555],[0,0,0,0],[8.999999E+09,8.999999E+09,8.999999E+09,8.999999E+09,8.999999E+09,8.999999E+09]];
    LOCAL CONST Robtarget Tr_meulage_motif_1_127 := [[-44.93175390625,69.35571875,64.22148828125],[0.363951430919515,-0.363241574410581,0.605870778174484,-0.607054787235555],[0,0,0,0],[8.999999E+09,8.999999E+09,8.999999E+09,8.999999E+09,8.999999E+09,8.999999E+09]];
    LOCAL CONST Robtarget Tr_meulage_motif_1_128 := [[-45.403390625,68.4739296875,64.22146484375],[0.363951430919515,-0.363241574410581,0.605870778174484,-0.607054787235555],[0,0,0,0],[8.999999E+09,8.999999E+09,8.999999E+09,8.999999E+09,8.999999E+09,8.999999E+09]];
    LOCAL CONST Robtarget Tr_meulage_motif_1_129 := [[-45.87502734375,67.5921328125,64.2214375],[0.363951430919515,-0.363241574410581,0.605870778174484,-0.607054787235555],[0,0,0,0],[8.999999E+09,8.999999E+09,8.999999E+09,8.999999E+09,8.999999E+09,8.999999E+09]];
    LOCAL CONST Robtarget Tr_meulage_motif_1_130 := [[-46.34666796875,66.71034375,64.2214140625],[0.363951430919515,-0.363241574410581,0.605870778174484,-0.607054787235555],[0,0,0,0],[8.999999E+09,8.999999E+09,8.999999E+09,8.999999E+09,8.999999E+09,8.999999E+09]];
    LOCAL CONST Robtarget Tr_meulage_motif_1_131 := [[-46.8183046875,65.828546875,64.22138671875],[0.363951430919515,-0.363241574410581,0.605870778174484,-0.607054787235555],[0,0,0,0],[8.999999E+09,8.999999E+09,8.999999E+09,8.999999E+09,8.999999E+09,8.999999E+09]];
    LOCAL CONST Robtarget Tr_meulage_motif_1_132 := [[-47.28994140625,64.9467578125,64.22136328125],[0.363951430919515,-0.363241574410581,0.605870778174484,-0.607054787235555],[0,0,0,0],[8.999999E+09,8.999999E+09,8.999999E+09,8.999999E+09,8.999999E+09,8.999999E+09]];
    LOCAL CONST Robtarget Tr_meulage_motif_1_133 := [[-47.761578125,64.06496484375,64.2213359375],[0.363951430919515,-0.363241574410581,0.605870778174484,-0.607054787235555],[0,0,0,0],[8.999999E+09,8.999999E+09,8.999999E+09,8.999999E+09,8.999999E+09,8.999999E+09]];
    LOCAL CONST Robtarget Tr_meulage_motif_1_134 := [[-48.23321875,63.183171875,64.2213125],[0.363951430919515,-0.363241574410581,0.605870778174484,-0.607054787235555],[0,0,0,0],[8.999999E+09,8.999999E+09,8.999999E+09,8.999999E+09,8.999999E+09,8.999999E+09]];
    LOCAL CONST Robtarget Tr_meulage_motif_1_135 := [[-48.70485546875,62.30137890625,64.2212890625],[0.363951430919515,-0.363241574410581,0.605870778174484,-0.607054787235555],[0,0,0,0],[8.999999E+09,8.999999E+09,8.999999E+09,8.999999E+09,8.999999E+09,8.999999E+09]];
    LOCAL CONST Robtarget Tr_meulage_motif_1_136 := [[-49.1764921875,61.4195859375,64.22126171875],[0.363951430919515,-0.363241574410581,0.605870778174484,-0.607054787235555],[0,0,0,0],[8.999999E+09,8.999999E+09,8.999999E+09,8.999999E+09,8.999999E+09,8.999999E+09]];
    LOCAL CONST Robtarget Tr_meulage_motif_1_137 := [[-49.64812890625,60.537796875,64.22123828125],[0.363951430919515,-0.363241574410581,0.605870778174484,-0.607054787235555],[0,0,0,0],[8.999999E+09,8.999999E+09,8.999999E+09,8.999999E+09,8.999999E+09,8.999999E+09]];
    LOCAL CONST Robtarget Tr_meulage_motif_1_138 := [[-50.109984375,59.65920703125,64.11084765625],[0.363951430919515,-0.363241574410581,0.605870778174484,-0.607054787235555],[0,0,0,0],[8.999999E+09,8.999999E+09,8.999999E+09,8.999999E+09,8.999999E+09,8.999999E+09]];
    LOCAL CONST Robtarget Tr_meulage_motif_1_139 := [[-50.54441015625,58.8181875,63.90007421875],[0.363951430919515,-0.363241574410581,0.605870778174484,-0.607054787235555],[0,0,0,0],[8.999999E+09,8.999999E+09,8.999999E+09,8.999999E+09,8.999999E+09,8.999999E+09]];
    LOCAL CONST Robtarget Tr_meulage_motif_1_140 := [[-50.93116015625,58.05802734375,63.6287734375],[0.363951430919515,-0.363241574410581,0.605870778174484,-0.607054787235555],[0,0,0,0],[8.999999E+09,8.999999E+09,8.999999E+09,8.999999E+09,8.999999E+09,8.999999E+09]];
    LOCAL CONST Robtarget Tr_meulage_motif_1_141 := [[-51.269203125,57.38837109375,63.35338671875],[0.363951430919515,-0.363241574410581,0.605870778174484,-0.607054787235555],[0,0,0,0],[8.999999E+09,8.999999E+09,8.999999E+09,8.999999E+09,8.999999E+09,8.999999E+09]];
    LOCAL CONST Robtarget Tr_meulage_motif_1_142 := [[-51.75355078125,56.39878515625,62.73851171875],[0.363951430919515,-0.363241574410581,0.605870778174484,-0.607054787235555],[0,0,0,0],[8.999999E+09,8.999999E+09,8.999999E+09,8.999999E+09,8.999999E+09,8.999999E+09]];
    LOCAL CONST Robtarget Tr_meulage_motif_1_143 := [[-52.188359375,55.4702421875,61.89258203125],[0.363951430919515,-0.363241574410581,0.605870778174484,-0.607054787235555],[0,0,0,0],[8.999999E+09,8.999999E+09,8.999999E+09,8.999999E+09,8.999999E+09,8.999999E+09]];
    LOCAL CONST Robtarget Tr_meulage_motif_1_144 := [[-52.53005859375,54.69174609375,60.87080859375],[0.363951430919515,-0.363241574410581,0.605870778174484,-0.607054787235555],[0,0,0,0],[8.999999E+09,8.999999E+09,8.999999E+09,8.999999E+09,8.999999E+09,8.999999E+09]];
    LOCAL CONST Robtarget Tr_meulage_motif_1_145 := [[-52.69696484375,54.227453125,59.75691796875],[0.363951430919515,-0.363241574410581,0.605870778174484,-0.607054787235555],[0,0,0,0],[8.999999E+09,8.999999E+09,8.999999E+09,8.999999E+09,8.999999E+09,8.999999E+09]];
    LOCAL CONST Robtarget Tr_meulage_motif_1_146 := [[-52.6702421875,54.1824921875,59.062390625],[0.363951430919515,-0.363241574410581,0.605870778174484,-0.607054787235555],[0,0,0,0],[8.999999E+09,8.999999E+09,8.999999E+09,8.999999E+09,8.999999E+09,8.999999E+09]];
    LOCAL CONST Robtarget Tr_meulage_motif_1_147 := [[-52.63273046875,54.1624453125,58.40251171875],[0.363951430919515,-0.363241574410581,0.605870778174484,-0.607054787235555],[0,0,0,0],[8.999999E+09,8.999999E+09,8.999999E+09,8.999999E+09,8.999999E+09,8.999999E+09]];
    LOCAL CONST Robtarget Tr_meulage_motif_1_148 := [[-52.56933984375,54.1907890625,57.7427890625],[0.363951430919515,-0.363241574410581,0.605870778174484,-0.607054787235555],[0,0,0,0],[8.999999E+09,8.999999E+09,8.999999E+09,8.999999E+09,8.999999E+09,8.999999E+09]];
    LOCAL CONST Robtarget Tr_meulage_motif_1_149 := [[-52.27185546875,54.59671484375,56.64333203125],[0.363951430919515,-0.363241574410581,0.605870778174484,-0.607054787235555],[0,0,0,0],[8.999999E+09,8.999999E+09,8.999999E+09,8.999999E+09,8.999999E+09,8.999999E+09]];
    LOCAL CONST Robtarget Tr_meulage_motif_1_150 := [[-51.81073046875,55.3215625,55.6388125],[0.363951430919515,-0.363241574410581,0.605870778174484,-0.607054787235555],[0,0,0,0],[8.999999E+09,8.999999E+09,8.999999E+09,8.999999E+09,8.999999E+09,8.999999E+09]];
    LOCAL CONST Robtarget Tr_meulage_motif_1_151 := [[-51.28102734375,56.1988671875,54.8116796875],[0.363951430919515,-0.363241574410581,0.605870778174484,-0.607054787235555],[0,0,0,0],[8.999999E+09,8.999999E+09,8.999999E+09,8.999999E+09,8.999999E+09,8.999999E+09]];
    LOCAL CONST Robtarget Tr_meulage_motif_1_152 := [[-50.934515625,56.7927421875,54.41676953125],[0.363951430919515,-0.363241574410581,0.605870778174484,-0.607054787235555],[0,0,0,0],[8.999999E+09,8.999999E+09,8.999999E+09,8.999999E+09,8.999999E+09,8.999999E+09]];
    LOCAL CONST Robtarget Tr_meulage_motif_1_153 := [[-50.360625,57.79921484375,53.93027734375],[0.363951430919515,-0.363241574410581,0.605870778174484,-0.607054787235555],[0,0,0,0],[8.999999E+09,8.999999E+09,8.999999E+09,8.999999E+09,8.999999E+09,8.999999E+09]];
    LOCAL CONST Robtarget Tr_meulage_motif_1_154 := [[-49.94709375,58.5363515625,53.66675],[0.363951430919515,-0.363241574410581,0.605870778174484,-0.607054787235555],[0,0,0,0],[8.999999E+09,8.999999E+09,8.999999E+09,8.999999E+09,8.999999E+09,8.999999E+09]];
    LOCAL CONST Robtarget Tr_meulage_motif_1_155 := [[-49.49592578125,59.351984375,53.4627265625],[0.363951430919515,-0.363241574410581,0.605870778174484,-0.607054787235555],[0,0,0,0],[8.999999E+09,8.999999E+09,8.999999E+09,8.999999E+09,8.999999E+09,8.999999E+09]];
    LOCAL CONST Robtarget Tr_meulage_motif_1_156 := [[-49.02682421875,60.2142265625,53.3543828125],[0.363951430919515,-0.363241574410581,0.605870778174484,-0.607054787235555],[0,0,0,0],[8.999999E+09,8.999999E+09,8.999999E+09,8.999999E+09,8.999999E+09,8.999999E+09]];
    LOCAL CONST Robtarget Tr_meulage_motif_1_157 := [[-48.552421875,61.08610546875,53.24404296875],[0.363951430919515,-0.363241574410581,0.605870778174484,-0.607054787235555],[0,0,0,0],[8.999999E+09,8.999999E+09,8.999999E+09,8.999999E+09,8.999999E+09,8.999999E+09]];
    LOCAL CONST Robtarget Tr_meulage_motif_1_158 := [[-48.08078125,61.9678984375,53.2440703125],[0.363951430919515,-0.363241574410581,0.605870778174484,-0.607054787235555],[0,0,0,0],[8.999999E+09,8.999999E+09,8.999999E+09,8.999999E+09,8.999999E+09,8.999999E+09]];
    LOCAL CONST Robtarget Tr_meulage_motif_1_159 := [[-47.60914453125,62.84969140625,53.24409375],[0.363951430919515,-0.363241574410581,0.605870778174484,-0.607054787235555],[0,0,0,0],[8.999999E+09,8.999999E+09,8.999999E+09,8.999999E+09,8.999999E+09,8.999999E+09]];
    LOCAL CONST Robtarget Tr_meulage_motif_1_160 := [[-47.1375078125,63.731484375,53.24412109375],[0.363951430919515,-0.363241574410581,0.605870778174484,-0.607054787235555],[0,0,0,0],[8.999999E+09,8.999999E+09,8.999999E+09,8.999999E+09,8.999999E+09,8.999999E+09]];
    LOCAL CONST Robtarget Tr_meulage_motif_1_161 := [[-46.66587109375,64.61327734375,53.24414453125],[0.363951430919515,-0.363241574410581,0.605870778174484,-0.607054787235555],[0,0,0,0],[8.999999E+09,8.999999E+09,8.999999E+09,8.999999E+09,8.999999E+09,8.999999E+09]];
    LOCAL CONST Robtarget Tr_meulage_motif_1_162 := [[-46.19423046875,65.4950703125,53.24416796875],[0.363951430919515,-0.363241574410581,0.605870778174484,-0.607054787235555],[0,0,0,0],[8.999999E+09,8.999999E+09,8.999999E+09,8.999999E+09,8.999999E+09,8.999999E+09]];
    LOCAL CONST Robtarget Tr_meulage_motif_1_163 := [[-45.72259375,66.376859375,53.2441953125],[0.363951430919515,-0.363241574410581,0.605870778174484,-0.607054787235555],[0,0,0,0],[8.999999E+09,8.999999E+09,8.999999E+09,8.999999E+09,8.999999E+09,8.999999E+09]];
    LOCAL CONST Robtarget Tr_meulage_motif_1_164 := [[-45.25095703125,67.25865625,53.24421875],[0.363951430919515,-0.363241574410581,0.605870778174484,-0.607054787235555],[0,0,0,0],[8.999999E+09,8.999999E+09,8.999999E+09,8.999999E+09,8.999999E+09,8.999999E+09]];
    LOCAL CONST Robtarget Tr_meulage_motif_1_165 := [[-44.7793203125,68.1404453125,53.24424609375],[0.363951430919515,-0.363241574410581,0.605870778174484,-0.607054787235555],[0,0,0,0],[8.999999E+09,8.999999E+09,8.999999E+09,8.999999E+09,8.999999E+09,8.999999E+09]];
    LOCAL CONST Robtarget Tr_meulage_motif_1_166 := [[-44.3076796875,69.0222421875,53.24426953125],[0.363951430919515,-0.363241574410581,0.605870778174484,-0.607054787235555],[0,0,0,0],[8.999999E+09,8.999999E+09,8.999999E+09,8.999999E+09,8.999999E+09,8.999999E+09]];
    LOCAL CONST Robtarget Tr_meulage_motif_1_167 := [[-43.83604296875,69.90403125,53.244296875],[0.363951430919515,-0.363241574410581,0.605870778174484,-0.607054787235555],[0,0,0,0],[8.999999E+09,8.999999E+09,8.999999E+09,8.999999E+09,8.999999E+09,8.999999E+09]];
    LOCAL CONST Robtarget Tr_meulage_motif_1_168 := [[-43.36440625,70.7858203125,53.2443203125],[0.363951430919515,-0.363241574410581,0.605870778174484,-0.607054787235555],[0,0,0,0],[8.999999E+09,8.999999E+09,8.999999E+09,8.999999E+09,8.999999E+09,8.999999E+09]];
    LOCAL CONST Robtarget Tr_meulage_motif_1_169 := [[-42.89276953125,71.6676171875,53.24434375],[0.363951430919515,-0.363241574410581,0.605870778174484,-0.607054787235555],[0,0,0,0],[8.999999E+09,8.999999E+09,8.999999E+09,8.999999E+09,8.999999E+09,8.999999E+09]];
    LOCAL CONST Robtarget Tr_meulage_motif_1_170 := [[-42.42112890625,72.54940625,53.24437109375],[0.363951430919515,-0.363241574410581,0.605870778174484,-0.607054787235555],[0,0,0,0],[8.999999E+09,8.999999E+09,8.999999E+09,8.999999E+09,8.999999E+09,8.999999E+09]];
    LOCAL CONST Robtarget Tr_meulage_motif_1_171 := [[-41.9494921875,73.431203125,53.24439453125],[0.363951430919515,-0.363241574410581,0.605870778174484,-0.607054787235555],[0,0,0,0],[8.999999E+09,8.999999E+09,8.999999E+09,8.999999E+09,8.999999E+09,8.999999E+09]];
    LOCAL CONST Robtarget Tr_meulage_motif_1_172 := [[-41.47785546875,74.3129921875,53.244421875],[0.363951430919515,-0.363241574410581,0.605870778174484,-0.607054787235555],[0,0,0,0],[8.999999E+09,8.999999E+09,8.999999E+09,8.999999E+09,8.999999E+09,8.999999E+09]];
    LOCAL CONST Robtarget Tr_meulage_motif_1_173 := [[-41.00621875,75.1947890625,53.2444453125],[0.363951430919515,-0.363241574410581,0.605870778174484,-0.607054787235555],[0,0,0,0],[8.999999E+09,8.999999E+09,8.999999E+09,8.999999E+09,8.999999E+09,8.999999E+09]];
    LOCAL CONST Robtarget Tr_meulage_motif_1_174 := [[-40.534578125,76.076578125,53.24447265625],[0.363951430919515,-0.363241574410581,0.605870778174484,-0.607054787235555],[0,0,0,0],[8.999999E+09,8.999999E+09,8.999999E+09,8.999999E+09,8.999999E+09,8.999999E+09]];
    LOCAL CONST Robtarget Tr_meulage_motif_1_175 := [[-40.06294140625,76.9583671875,53.24449609375],[0.363951430919515,-0.363241574410581,0.605870778174484,-0.607054787235555],[0,0,0,0],[8.999999E+09,8.999999E+09,8.999999E+09,8.999999E+09,8.999999E+09,8.999999E+09]];
    LOCAL CONST Robtarget Tr_meulage_motif_1_176 := [[-39.5913046875,77.8401640625,53.2445234375],[0.363951430919515,-0.363241574410581,0.605870778174484,-0.607054787235555],[0,0,0,0],[8.999999E+09,8.999999E+09,8.999999E+09,8.999999E+09,8.999999E+09,8.999999E+09]];
    LOCAL CONST Robtarget Tr_meulage_motif_1_177 := [[-39.11966796875,78.721953125,53.244546875],[0.363951430919515,-0.363241574410581,0.605870778174484,-0.607054787235555],[0,0,0,0],[8.999999E+09,8.999999E+09,8.999999E+09,8.999999E+09,8.999999E+09,8.999999E+09]];
    LOCAL CONST Robtarget Tr_meulage_motif_1_178 := [[-38.64802734375,79.60375,53.2445703125],[0.363951430919515,-0.363241574410581,0.605870778174484,-0.607054787235555],[0,0,0,0],[8.999999E+09,8.999999E+09,8.999999E+09,8.999999E+09,8.999999E+09,8.999999E+09]];
    LOCAL CONST Robtarget Tr_meulage_motif_1_179 := [[-38.176390625,80.4855390625,53.24459765625],[0.363951430919515,-0.363241574410581,0.605870778174484,-0.607054787235555],[0,0,0,0],[8.999999E+09,8.999999E+09,8.999999E+09,8.999999E+09,8.999999E+09,8.999999E+09]];
    LOCAL CONST Robtarget Tr_meulage_motif_1_180 := [[-37.70475390625,81.3673359375,53.24462109375],[0.363951430919515,-0.363241574410581,0.605870778174484,-0.607054787235555],[0,0,0,0],[8.999999E+09,8.999999E+09,8.999999E+09,8.999999E+09,8.999999E+09,8.999999E+09]];
    LOCAL CONST Robtarget Tr_meulage_motif_1_181 := [[-37.2331171875,82.249125,53.2446484375],[0.363951430919515,-0.363241574410581,0.605870778174484,-0.607054787235555],[0,0,0,0],[8.999999E+09,8.999999E+09,8.999999E+09,8.999999E+09,8.999999E+09,8.999999E+09]];
    LOCAL CONST Robtarget Tr_meulage_motif_1_182 := [[-36.7614765625,83.130921875,53.244671875],[0.363951430919515,-0.363241574410581,0.605870778174484,-0.607054787235555],[0,0,0,0],[8.999999E+09,8.999999E+09,8.999999E+09,8.999999E+09,8.999999E+09,8.999999E+09]];
    LOCAL CONST Robtarget Tr_meulage_motif_1_183 := [[-36.28983984375,84.0127109375,53.24469921875],[0.363951430919515,-0.363241574410581,0.605870778174484,-0.607054787235555],[0,0,0,0],[8.999999E+09,8.999999E+09,8.999999E+09,8.999999E+09,8.999999E+09,8.999999E+09]];
    LOCAL CONST Robtarget Tr_meulage_motif_1_184 := [[-35.818203125,84.8945,53.24472265625],[0.363951430919515,-0.363241574410581,0.605870778174484,-0.607054787235555],[0,0,0,0],[8.999999E+09,8.999999E+09,8.999999E+09,8.999999E+09,8.999999E+09,8.999999E+09]];
    LOCAL CONST Robtarget Tr_meulage_motif_1_185 := [[-35.34656640625,85.776296875,53.24474609375],[0.363951430919515,-0.363241574410581,0.605870778174484,-0.607054787235555],[0,0,0,0],[8.999999E+09,8.999999E+09,8.999999E+09,8.999999E+09,8.999999E+09,8.999999E+09]];
    LOCAL CONST Robtarget Tr_meulage_motif_1_186 := [[-34.87492578125,86.6580859375,53.2447734375],[0.363951430919515,-0.363241574410581,0.605870778174484,-0.607054787235555],[0,0,0,0],[8.999999E+09,8.999999E+09,8.999999E+09,8.999999E+09,8.999999E+09,8.999999E+09]];
    LOCAL CONST Robtarget Tr_meulage_motif_1_187 := [[-34.4032890625,87.5398828125,53.244796875],[0.363951430919515,-0.363241574410581,0.605870778174484,-0.607054787235555],[0,0,0,0],[8.999999E+09,8.999999E+09,8.999999E+09,8.999999E+09,8.999999E+09,8.999999E+09]];
    LOCAL CONST Robtarget Tr_meulage_motif_1_188 := [[-33.92888671875,88.4117578125,53.13445703125],[0.363951430919515,-0.363241574410581,0.605870778174484,-0.607054787235555],[0,0,0,0],[8.999999E+09,8.999999E+09,8.999999E+09,8.999999E+09,8.999999E+09,8.999999E+09]];
    LOCAL CONST Robtarget Tr_meulage_motif_1_189 := [[-33.4705,89.2399765625,52.92373046875],[0.363951430919515,-0.363241574410581,0.605870778174484,-0.607054787235555],[0,0,0,0],[8.999999E+09,8.999999E+09,8.999999E+09,8.999999E+09,8.999999E+09,8.999999E+09]];
    LOCAL CONST Robtarget Tr_meulage_motif_1_190 := [[-33.05290234375,89.98365625,52.65247265625],[0.363951430919515,-0.363241574410581,0.605870778174484,-0.607054787235555],[0,0,0,0],[8.999999E+09,8.999999E+09,8.999999E+09,8.999999E+09,8.999999E+09,8.999999E+09]];
    LOCAL CONST Robtarget Tr_meulage_motif_1_191 := [[-32.700076171875,90.601828125,52.34898046875],[0.363951430919515,-0.363241574410581,0.605870778174484,-0.607054787235555],[0,0,0,0],[8.999999E+09,8.999999E+09,8.999999E+09,8.999999E+09,8.999999E+09,8.999999E+09]];
    LOCAL CONST Robtarget Tr_meulage_motif_1_192 := [[-32.17459375,91.4939296875,51.68784765625],[0.363951430919515,-0.363241574410581,0.605870778174484,-0.607054787235555],[0,0,0,0],[8.999999E+09,8.999999E+09,8.999999E+09,8.999999E+09,8.999999E+09,8.999999E+09]];
    LOCAL CONST Robtarget Tr_meulage_motif_1_193 := [[-31.69803515625,92.26190625,50.78778515625],[0.363951430919515,-0.363241574410581,0.605870778174484,-0.607054787235555],[0,0,0,0],[8.999999E+09,8.999999E+09,8.999999E+09,8.999999E+09,8.999999E+09,8.999999E+09]];
    LOCAL CONST Robtarget Tr_meulage_motif_1_194 := [[-31.38637890625,92.7019296875,49.74394921875],[0.363951430919515,-0.363241574410581,0.605870778174484,-0.607054787235555],[0,0,0,0],[8.999999E+09,8.999999E+09,8.999999E+09,8.999999E+09,8.999999E+09,8.999999E+09]];
    LOCAL CONST Robtarget Tr_meulage_motif_1_195 := [[-31.2598984375,92.8438515625,49.05215234375],[0.363951430919515,-0.363241574410581,0.605870778174484,-0.607054787235555],[0,0,0,0],[8.999999E+09,8.999999E+09,8.999999E+09,8.999999E+09,8.999999E+09,8.999999E+09]];
    LOCAL CONST Robtarget Tr_meulage_motif_1_196 := [[-31.186103515625,92.8768046875,48.28375],[0.363951430919515,-0.363241574410581,0.605870778174484,-0.607054787235555],[0,0,0,0],[8.999999E+09,8.999999E+09,8.999999E+09,8.999999E+09,8.999999E+09,8.999999E+09]];
    LOCAL CONST Robtarget Tr_meulage_motif_1_197 := [[-31.17399609375,92.7944375,47.515484375],[0.363951430919515,-0.363241574410581,0.605870778174484,-0.607054787235555],[0,0,0,0],[8.999999E+09,8.999999E+09,8.999999E+09,8.999999E+09,8.999999E+09,8.999999E+09]];
    LOCAL CONST Robtarget Tr_meulage_motif_1_198 := [[-31.309017578125,92.39084375,46.40951953125],[0.363951430919515,-0.363241574410581,0.605870778174484,-0.607054787235555],[0,0,0,0],[8.999999E+09,8.999999E+09,8.999999E+09,8.999999E+09,8.999999E+09,8.999999E+09]];
    LOCAL CONST Robtarget Tr_meulage_motif_1_199 := [[-31.471193359375,92.0077578125,45.82503515625],[0.363951430919515,-0.363241574410581,0.605870778174484,-0.607054787235555],[0,0,0,0],[8.999999E+09,8.999999E+09,8.999999E+09,8.999999E+09,8.999999E+09,8.999999E+09]];
    LOCAL CONST Robtarget Tr_meulage_motif_1_200 := [[-31.839263671875,91.1986015625,44.93969140625],[0.363951430919515,-0.363241574410581,0.605870778174484,-0.607054787235555],[0,0,0,0],[8.999999E+09,8.999999E+09,8.999999E+09,8.999999E+09,8.999999E+09,8.999999E+09]];
    LOCAL CONST Robtarget Tr_meulage_motif_1_201 := [[-32.0919921875,90.6695859375,44.52625390625],[0.363951430919515,-0.363241574410581,0.605870778174484,-0.607054787235555],[0,0,0,0],[8.999999E+09,8.999999E+09,8.999999E+09,8.999999E+09,8.999999E+09,8.999999E+09]];
    LOCAL CONST Robtarget Tr_meulage_motif_1_202 := [[-32.588369140625,89.667328125,43.9832265625],[0.363951430919515,-0.363241574410581,0.605870778174484,-0.607054787235555],[0,0,0,0],[8.999999E+09,8.999999E+09,8.999999E+09,8.999999E+09,8.999999E+09,8.999999E+09]];
    LOCAL CONST Robtarget Tr_meulage_motif_1_203 := [[-32.960984375,88.9303671875,43.6883203125],[0.363951430919515,-0.363241574410581,0.605870778174484,-0.607054787235555],[0,0,0,0],[8.999999E+09,8.999999E+09,8.999999E+09,8.999999E+09,8.999999E+09,8.999999E+09]];
    LOCAL CONST Robtarget Tr_meulage_motif_1_204 := [[-33.38894921875,88.1023359375,43.484234375],[0.363951430919515,-0.363241574410581,0.605870778174484,-0.607054787235555],[0,0,0,0],[8.999999E+09,8.999999E+09,8.999999E+09,8.999999E+09,8.999999E+09,8.999999E+09]];
    LOCAL CONST Robtarget Tr_meulage_motif_1_205 := [[-33.845734375,87.2335078125,43.37588671875],[0.363951430919515,-0.363241574410581,0.605870778174484,-0.607054787235555],[0,0,0,0],[8.999999E+09,8.999999E+09,8.999999E+09,8.999999E+09,8.999999E+09,8.999999E+09]];
    LOCAL CONST Robtarget Tr_meulage_motif_1_206 := [[-34.30758984375,86.354921875,43.265484375],[0.363951430919515,-0.363241574410581,0.605870778174484,-0.607054787235555],[0,0,0,0],[8.999999E+09,8.999999E+09,8.999999E+09,8.999999E+09,8.999999E+09,8.999999E+09]];
    LOCAL CONST Robtarget Tr_meulage_motif_1_207 := [[-34.7792265625,85.4731328125,43.26545703125],[0.363951430919515,-0.363241574410581,0.605870778174484,-0.607054787235555],[0,0,0,0],[8.999999E+09,8.999999E+09,8.999999E+09,8.999999E+09,8.999999E+09,8.999999E+09]];
    LOCAL CONST Robtarget Tr_meulage_motif_1_208 := [[-35.25086328125,84.5913359375,43.26543359375],[0.363951430919515,-0.363241574410581,0.605870778174484,-0.607054787235555],[0,0,0,0],[8.999999E+09,8.999999E+09,8.999999E+09,8.999999E+09,8.999999E+09,8.999999E+09]];
    LOCAL CONST Robtarget Tr_meulage_motif_1_209 := [[-35.7225,83.709546875,43.26540625],[0.363951430919515,-0.363241574410581,0.605870778174484,-0.607054787235555],[0,0,0,0],[8.999999E+09,8.999999E+09,8.999999E+09,8.999999E+09,8.999999E+09,8.999999E+09]];
    LOCAL CONST Robtarget Tr_meulage_motif_1_210 := [[-36.194140625,82.8277578125,43.2653828125],[0.363951430919515,-0.363241574410581,0.605870778174484,-0.607054787235555],[0,0,0,0],[8.999999E+09,8.999999E+09,8.999999E+09,8.999999E+09,8.999999E+09,8.999999E+09]];
    LOCAL CONST Robtarget Tr_meulage_motif_1_211 := [[-36.66577734375,81.9459609375,43.265359375],[0.363951430919515,-0.363241574410581,0.605870778174484,-0.607054787235555],[0,0,0,0],[8.999999E+09,8.999999E+09,8.999999E+09,8.999999E+09,8.999999E+09,8.999999E+09]];
    LOCAL CONST Robtarget Tr_meulage_motif_1_212 := [[-37.1374140625,81.064171875,43.26533203125],[0.363951430919515,-0.363241574410581,0.605870778174484,-0.607054787235555],[0,0,0,0],[8.999999E+09,8.999999E+09,8.999999E+09,8.999999E+09,8.999999E+09,8.999999E+09]];
    LOCAL CONST Robtarget Tr_meulage_motif_1_213 := [[-37.60905078125,80.182375,43.26530859375],[0.363951430919515,-0.363241574410581,0.605870778174484,-0.607054787235555],[0,0,0,0],[8.999999E+09,8.999999E+09,8.999999E+09,8.999999E+09,8.999999E+09,8.999999E+09]];
    LOCAL CONST Robtarget Tr_meulage_motif_1_214 := [[-38.08069140625,79.3005859375,43.26528125],[0.363951430919515,-0.363241574410581,0.605870778174484,-0.607054787235555],[0,0,0,0],[8.999999E+09,8.999999E+09,8.999999E+09,8.999999E+09,8.999999E+09,8.999999E+09]];
    LOCAL CONST Robtarget Tr_meulage_motif_1_215 := [[-38.552328125,78.4187890625,43.2652578125],[0.363951430919515,-0.363241574410581,0.605870778174484,-0.607054787235555],[0,0,0,0],[8.999999E+09,8.999999E+09,8.999999E+09,8.999999E+09,8.999999E+09,8.999999E+09]];
    LOCAL CONST Robtarget Tr_meulage_motif_1_216 := [[-39.02396484375,77.537,43.26523046875],[0.363951430919515,-0.363241574410581,0.605870778174484,-0.607054787235555],[0,0,0,0],[8.999999E+09,8.999999E+09,8.999999E+09,8.999999E+09,8.999999E+09,8.999999E+09]];
    LOCAL CONST Robtarget Tr_meulage_motif_1_217 := [[-39.4956015625,76.6552109375,43.26520703125],[0.363951430919515,-0.363241574410581,0.605870778174484,-0.607054787235555],[0,0,0,0],[8.999999E+09,8.999999E+09,8.999999E+09,8.999999E+09,8.999999E+09,8.999999E+09]];
    LOCAL CONST Robtarget Tr_meulage_motif_1_218 := [[-39.9672421875,75.7734140625,43.26518359375],[0.363951430919515,-0.363241574410581,0.605870778174484,-0.607054787235555],[0,0,0,0],[8.999999E+09,8.999999E+09,8.999999E+09,8.999999E+09,8.999999E+09,8.999999E+09]];
    LOCAL CONST Robtarget Tr_meulage_motif_1_219 := [[-40.43887890625,74.891625,43.26515625],[0.363951430919515,-0.363241574410581,0.605870778174484,-0.607054787235555],[0,0,0,0],[8.999999E+09,8.999999E+09,8.999999E+09,8.999999E+09,8.999999E+09,8.999999E+09]];
    LOCAL CONST Robtarget Tr_meulage_motif_1_220 := [[-40.910515625,74.009828125,43.2651328125],[0.363951430919515,-0.363241574410581,0.605870778174484,-0.607054787235555],[0,0,0,0],[8.999999E+09,8.999999E+09,8.999999E+09,8.999999E+09,8.999999E+09,8.999999E+09]];
    LOCAL CONST Robtarget Tr_meulage_motif_1_221 := [[-41.38215234375,73.1280390625,43.26510546875],[0.363951430919515,-0.363241574410581,0.605870778174484,-0.607054787235555],[0,0,0,0],[8.999999E+09,8.999999E+09,8.999999E+09,8.999999E+09,8.999999E+09,8.999999E+09]];
    LOCAL CONST Robtarget Tr_meulage_motif_1_222 := [[-41.85379296875,72.2462421875,43.26508203125],[0.363951430919515,-0.363241574410581,0.605870778174484,-0.607054787235555],[0,0,0,0],[8.999999E+09,8.999999E+09,8.999999E+09,8.999999E+09,8.999999E+09,8.999999E+09]];
    LOCAL CONST Robtarget Tr_meulage_motif_1_223 := [[-42.3254296875,71.364453125,43.2650546875],[0.363951430919515,-0.363241574410581,0.605870778174484,-0.607054787235555],[0,0,0,0],[8.999999E+09,8.999999E+09,8.999999E+09,8.999999E+09,8.999999E+09,8.999999E+09]];
    LOCAL CONST Robtarget Tr_meulage_motif_1_224 := [[-42.79706640625,70.4826640625,43.26503125],[0.363951430919515,-0.363241574410581,0.605870778174484,-0.607054787235555],[0,0,0,0],[8.999999E+09,8.999999E+09,8.999999E+09,8.999999E+09,8.999999E+09,8.999999E+09]];
    LOCAL CONST Robtarget Tr_meulage_motif_1_225 := [[-43.268703125,69.6008671875,43.26500390625],[0.363951430919515,-0.363241574410581,0.605870778174484,-0.607054787235555],[0,0,0,0],[8.999999E+09,8.999999E+09,8.999999E+09,8.999999E+09,8.999999E+09,8.999999E+09]];
    LOCAL CONST Robtarget Tr_meulage_motif_1_226 := [[-43.74034375,68.719078125,43.26498046875],[0.363951430919515,-0.363241574410581,0.605870778174484,-0.607054787235555],[0,0,0,0],[8.999999E+09,8.999999E+09,8.999999E+09,8.999999E+09,8.999999E+09,8.999999E+09]];
    LOCAL CONST Robtarget Tr_meulage_motif_1_227 := [[-44.21198046875,67.83728125,43.26495703125],[0.363951430919515,-0.363241574410581,0.605870778174484,-0.607054787235555],[0,0,0,0],[8.999999E+09,8.999999E+09,8.999999E+09,8.999999E+09,8.999999E+09,8.999999E+09]];
    LOCAL CONST Robtarget Tr_meulage_motif_1_228 := [[-44.6836171875,66.9554921875,43.2649296875],[0.363951430919515,-0.363241574410581,0.605870778174484,-0.607054787235555],[0,0,0,0],[8.999999E+09,8.999999E+09,8.999999E+09,8.999999E+09,8.999999E+09,8.999999E+09]];
    LOCAL CONST Robtarget Tr_meulage_motif_1_229 := [[-45.15525390625,66.0736953125,43.26490625],[0.363951430919515,-0.363241574410581,0.605870778174484,-0.607054787235555],[0,0,0,0],[8.999999E+09,8.999999E+09,8.999999E+09,8.999999E+09,8.999999E+09,8.999999E+09]];
    LOCAL CONST Robtarget Tr_meulage_motif_1_230 := [[-45.62689453125,65.19190625,43.26487890625],[0.363951430919515,-0.363241574410581,0.605870778174484,-0.607054787235555],[0,0,0,0],[8.999999E+09,8.999999E+09,8.999999E+09,8.999999E+09,8.999999E+09,8.999999E+09]];
    LOCAL CONST Robtarget Tr_meulage_motif_1_231 := [[-46.09853125,64.31011328125,43.26485546875],[0.363951430919515,-0.363241574410581,0.605870778174484,-0.607054787235555],[0,0,0,0],[8.999999E+09,8.999999E+09,8.999999E+09,8.999999E+09,8.999999E+09,8.999999E+09]];
    LOCAL CONST Robtarget Tr_meulage_motif_1_232 := [[-46.57016796875,63.4283203125,43.264828125],[0.363951430919515,-0.363241574410581,0.605870778174484,-0.607054787235555],[0,0,0,0],[8.999999E+09,8.999999E+09,8.999999E+09,8.999999E+09,8.999999E+09,8.999999E+09]];
    LOCAL CONST Robtarget Tr_meulage_motif_1_233 := [[-47.0418046875,62.54652734375,43.2648046875],[0.363951430919515,-0.363241574410581,0.605870778174484,-0.607054787235555],[0,0,0,0],[8.999999E+09,8.999999E+09,8.999999E+09,8.999999E+09,8.999999E+09,8.999999E+09]];
    LOCAL CONST Robtarget Tr_meulage_motif_1_234 := [[-47.5134453125,61.664734375,43.26478125],[0.363951430919515,-0.363241574410581,0.605870778174484,-0.607054787235555],[0,0,0,0],[8.999999E+09,8.999999E+09,8.999999E+09,8.999999E+09,8.999999E+09,8.999999E+09]];
    LOCAL CONST Robtarget Tr_meulage_motif_1_235 := [[-47.98508203125,60.7829453125,43.26475390625],[0.363951430919515,-0.363241574410581,0.605870778174484,-0.607054787235555],[0,0,0,0],[8.999999E+09,8.999999E+09,8.999999E+09,8.999999E+09,8.999999E+09,8.999999E+09]];
    LOCAL CONST Robtarget Tr_meulage_motif_1_236 := [[-48.45671875,59.90115234375,43.26473046875],[0.363951430919515,-0.363241574410581,0.605870778174484,-0.607054787235555],[0,0,0,0],[8.999999E+09,8.999999E+09,8.999999E+09,8.999999E+09,8.999999E+09,8.999999E+09]];
    LOCAL CONST Robtarget Tr_meulage_motif_1_237 := [[-48.91857421875,59.0225625,43.15432421875],[0.363951430919515,-0.363241574410581,0.605870778174484,-0.607054787235555],[0,0,0,0],[8.999999E+09,8.999999E+09,8.999999E+09,8.999999E+09,8.999999E+09,8.999999E+09]];
    LOCAL CONST Robtarget Tr_meulage_motif_1_238 := [[-49.35299609375,58.18154296875,42.94355078125],[0.363951430919515,-0.363241574410581,0.605870778174484,-0.607054787235555],[0,0,0,0],[8.999999E+09,8.999999E+09,8.999999E+09,8.999999E+09,8.999999E+09,8.999999E+09]];
    LOCAL CONST Robtarget Tr_meulage_motif_1_239 := [[-49.73975,57.4213828125,42.672265625],[0.363951430919515,-0.363241574410581,0.605870778174484,-0.607054787235555],[0,0,0,0],[8.999999E+09,8.999999E+09,8.999999E+09,8.999999E+09,8.999999E+09,8.999999E+09]];
    LOCAL CONST Robtarget Tr_meulage_motif_1_240 := [[-50.05806640625,56.784765625,42.368734375],[0.363951430919515,-0.363241574410581,0.605870778174484,-0.607054787235555],[0,0,0,0],[8.999999E+09,8.999999E+09,8.999999E+09,8.999999E+09,8.999999E+09,8.999999E+09]];
    LOCAL CONST Robtarget Tr_meulage_motif_1_241 := [[-50.50837109375,55.85249609375,41.70755078125],[0.363951430919515,-0.363241574410581,0.605870778174484,-0.607054787235555],[0,0,0,0],[8.999999E+09,8.999999E+09,8.999999E+09,8.999999E+09,8.999999E+09,8.999999E+09]];
    LOCAL CONST Robtarget Tr_meulage_motif_1_242 := [[-50.8384375,55.10721875,40.7696953125],[0.363951430919515,-0.363241574410581,0.605870778174484,-0.607054787235555],[0,0,0,0],[8.999999E+09,8.999999E+09,8.999999E+09,8.999999E+09,8.999999E+09,8.999999E+09]];
    LOCAL CONST Robtarget Tr_meulage_motif_1_243 := [[-50.9481328125,54.766234375,39.775390625],[0.363951430919515,-0.363241574410581,0.605870778174484,-0.607054787235555],[0,0,0,0],[8.999999E+09,8.999999E+09,8.999999E+09,8.999999E+09,8.999999E+09,8.999999E+09]];
    LOCAL CONST Robtarget Tr_meulage_motif_1_244 := [[-50.90251171875,54.77548046875,39.219],[0.363951430919515,-0.363241574410581,0.605870778174484,-0.607054787235555],[0,0,0,0],[8.999999E+09,8.999999E+09,8.999999E+09,8.999999E+09,8.999999E+09,8.999999E+09]];
    LOCAL CONST Robtarget Tr_meulage_motif_1_245 := [[-50.88083984375,54.75901171875,38.80195703125],[0.363951430919515,-0.363241574410581,0.605870778174484,-0.607054787235555],[0,0,0,0],[8.999999E+09,8.999999E+09,8.999999E+09,8.999999E+09,8.999999E+09,8.999999E+09]];
    LOCAL CONST Robtarget Tr_meulage_motif_1_246 := [[-50.6550390625,55.04896875,37.83464453125],[0.363951430919515,-0.363241574410581,0.605870778174484,-0.607054787235555],[0,0,0,0],[8.999999E+09,8.999999E+09,8.999999E+09,8.999999E+09,8.999999E+09,8.999999E+09]];
    LOCAL CONST Robtarget Tr_meulage_motif_1_247 := [[-50.21531640625,55.74592578125,36.91887890625],[0.363951430919515,-0.363241574410581,0.605870778174484,-0.607054787235555],[0,0,0,0],[8.999999E+09,8.999999E+09,8.999999E+09,8.999999E+09,8.999999E+09,8.999999E+09]];
    LOCAL CONST Robtarget Tr_meulage_motif_1_248 := [[-49.902609375,56.27290234375,36.49687890625],[0.363951430919515,-0.363241574410581,0.605870778174484,-0.607054787235555],[0,0,0,0],[8.999999E+09,8.999999E+09,8.999999E+09,8.999999E+09,8.999999E+09,8.999999E+09]];
    LOCAL CONST Robtarget Tr_meulage_motif_1_249 := [[-49.33941796875,57.2535234375,35.9675546875],[0.363951430919515,-0.363241574410581,0.605870778174484,-0.607054787235555],[0,0,0,0],[8.999999E+09,8.999999E+09,8.999999E+09,8.999999E+09,8.999999E+09,8.999999E+09]];
    LOCAL CONST Robtarget Tr_meulage_motif_1_250 := [[-48.9258828125,57.99065625,35.70401171875],[0.363951430919515,-0.363241574410581,0.605870778174484,-0.607054787235555],[0,0,0,0],[8.999999E+09,8.999999E+09,8.999999E+09,8.999999E+09,8.999999E+09,8.999999E+09]];
    LOCAL CONST Robtarget Tr_meulage_motif_1_251 := [[-48.47471484375,58.8062890625,35.4999765625],[0.363951430919515,-0.363241574410581,0.605870778174484,-0.607054787235555],[0,0,0,0],[8.999999E+09,8.999999E+09,8.999999E+09,8.999999E+09,8.999999E+09,8.999999E+09]];
    LOCAL CONST Robtarget Tr_meulage_motif_1_252 := [[-48.0056171875,59.66853125,35.3916796875],[0.363951430919515,-0.363241574410581,0.605870778174484,-0.607054787235555],[0,0,0,0],[8.999999E+09,8.999999E+09,8.999999E+09,8.999999E+09,8.999999E+09,8.999999E+09]];
    LOCAL CONST Robtarget Tr_meulage_motif_1_253 := [[-47.5312109375,60.5404140625,35.28132421875],[0.363951430919515,-0.363241574410581,0.605870778174484,-0.607054787235555],[0,0,0,0],[8.999999E+09,8.999999E+09,8.999999E+09,8.999999E+09,8.999999E+09,8.999999E+09]];
    LOCAL CONST Robtarget Tr_meulage_motif_1_254 := [[-47.05957421875,61.422203125,35.28134765625],[0.363951430919515,-0.363241574410581,0.605870778174484,-0.607054787235555],[0,0,0,0],[8.999999E+09,8.999999E+09,8.999999E+09,8.999999E+09,8.999999E+09,8.999999E+09]];
    LOCAL CONST Robtarget Tr_meulage_motif_1_255 := [[-46.58793359375,62.30399609375,35.281375],[0.363951430919515,-0.363241574410581,0.605870778174484,-0.607054787235555],[0,0,0,0],[8.999999E+09,8.999999E+09,8.999999E+09,8.999999E+09,8.999999E+09,8.999999E+09]];
    LOCAL CONST Robtarget Tr_meulage_motif_1_256 := [[-46.116296875,63.1857890625,35.2813984375],[0.363951430919515,-0.363241574410581,0.605870778174484,-0.607054787235555],[0,0,0,0],[8.999999E+09,8.999999E+09,8.999999E+09,8.999999E+09,8.999999E+09,8.999999E+09]];
    LOCAL CONST Robtarget Tr_meulage_motif_1_257 := [[-45.64466015625,64.06758203125,35.281421875],[0.363951430919515,-0.363241574410581,0.605870778174484,-0.607054787235555],[0,0,0,0],[8.999999E+09,8.999999E+09,8.999999E+09,8.999999E+09,8.999999E+09,8.999999E+09]];
    LOCAL CONST Robtarget Tr_meulage_motif_1_258 := [[-45.1730234375,64.949375,35.28144921875],[0.363951430919515,-0.363241574410581,0.605870778174484,-0.607054787235555],[0,0,0,0],[8.999999E+09,8.999999E+09,8.999999E+09,8.999999E+09,8.999999E+09,8.999999E+09]];
    LOCAL CONST Robtarget Tr_meulage_motif_1_259 := [[-44.7013828125,65.8311640625,35.28147265625],[0.363951430919515,-0.363241574410581,0.605870778174484,-0.607054787235555],[0,0,0,0],[8.999999E+09,8.999999E+09,8.999999E+09,8.999999E+09,8.999999E+09,8.999999E+09]];
    LOCAL CONST Robtarget Tr_meulage_motif_1_260 := [[-44.22974609375,66.7129609375,35.2815],[0.363951430919515,-0.363241574410581,0.605870778174484,-0.607054787235555],[0,0,0,0],[8.999999E+09,8.999999E+09,8.999999E+09,8.999999E+09,8.999999E+09,8.999999E+09]];
    LOCAL CONST Robtarget Tr_meulage_motif_1_261 := [[-43.758109375,67.59475,35.2815234375],[0.363951430919515,-0.363241574410581,0.605870778174484,-0.607054787235555],[0,0,0,0],[8.999999E+09,8.999999E+09,8.999999E+09,8.999999E+09,8.999999E+09,8.999999E+09]];
    LOCAL CONST Robtarget Tr_meulage_motif_1_262 := [[-43.28647265625,68.476546875,35.28155078125],[0.363951430919515,-0.363241574410581,0.605870778174484,-0.607054787235555],[0,0,0,0],[8.999999E+09,8.999999E+09,8.999999E+09,8.999999E+09,8.999999E+09,8.999999E+09]];
    LOCAL CONST Robtarget Tr_meulage_motif_1_263 := [[-42.81483203125,69.3583359375,35.28157421875],[0.363951430919515,-0.363241574410581,0.605870778174484,-0.607054787235555],[0,0,0,0],[8.999999E+09,8.999999E+09,8.999999E+09,8.999999E+09,8.999999E+09,8.999999E+09]];
    LOCAL CONST Robtarget Tr_meulage_motif_1_264 := [[-42.3431953125,70.2401328125,35.28159765625],[0.363951430919515,-0.363241574410581,0.605870778174484,-0.607054787235555],[0,0,0,0],[8.999999E+09,8.999999E+09,8.999999E+09,8.999999E+09,8.999999E+09,8.999999E+09]];
    LOCAL CONST Robtarget Tr_meulage_motif_1_265 := [[-41.87155859375,71.121921875,35.281625],[0.363951430919515,-0.363241574410581,0.605870778174484,-0.607054787235555],[0,0,0,0],[8.999999E+09,8.999999E+09,8.999999E+09,8.999999E+09,8.999999E+09,8.999999E+09]];
    LOCAL CONST Robtarget Tr_meulage_motif_1_266 := [[-41.399921875,72.0037109375,35.2816484375],[0.363951430919515,-0.363241574410581,0.605870778174484,-0.607054787235555],[0,0,0,0],[8.999999E+09,8.999999E+09,8.999999E+09,8.999999E+09,8.999999E+09,8.999999E+09]];
    LOCAL CONST Robtarget Tr_meulage_motif_1_267 := [[-40.92828125,72.8855078125,35.28167578125],[0.363951430919515,-0.363241574410581,0.605870778174484,-0.607054787235555],[0,0,0,0],[8.999999E+09,8.999999E+09,8.999999E+09,8.999999E+09,8.999999E+09,8.999999E+09]];
    LOCAL CONST Robtarget Tr_meulage_motif_1_268 := [[-40.45664453125,73.767296875,35.28169921875],[0.363951430919515,-0.363241574410581,0.605870778174484,-0.607054787235555],[0,0,0,0],[8.999999E+09,8.999999E+09,8.999999E+09,8.999999E+09,8.999999E+09,8.999999E+09]];
    LOCAL CONST Robtarget Tr_meulage_motif_1_269 := [[-39.9850078125,74.64909375,35.2817265625],[0.363951430919515,-0.363241574410581,0.605870778174484,-0.607054787235555],[0,0,0,0],[8.999999E+09,8.999999E+09,8.999999E+09,8.999999E+09,8.999999E+09,8.999999E+09]];
    LOCAL CONST Robtarget Tr_meulage_motif_1_270 := [[-39.51337109375,75.5308828125,35.28175],[0.363951430919515,-0.363241574410581,0.605870778174484,-0.607054787235555],[0,0,0,0],[8.999999E+09,8.999999E+09,8.999999E+09,8.999999E+09,8.999999E+09,8.999999E+09]];
    LOCAL CONST Robtarget Tr_meulage_motif_1_271 := [[-39.04173046875,76.4126796875,35.2817734375],[0.363951430919515,-0.363241574410581,0.605870778174484,-0.607054787235555],[0,0,0,0],[8.999999E+09,8.999999E+09,8.999999E+09,8.999999E+09,8.999999E+09,8.999999E+09]];
    LOCAL CONST Robtarget Tr_meulage_motif_1_272 := [[-38.57009375,77.29446875,35.28180078125],[0.363951430919515,-0.363241574410581,0.605870778174484,-0.607054787235555],[0,0,0,0],[8.999999E+09,8.999999E+09,8.999999E+09,8.999999E+09,8.999999E+09,8.999999E+09]];
    LOCAL CONST Robtarget Tr_meulage_motif_1_273 := [[-38.09845703125,78.1762578125,35.28182421875],[0.363951430919515,-0.363241574410581,0.605870778174484,-0.607054787235555],[0,0,0,0],[8.999999E+09,8.999999E+09,8.999999E+09,8.999999E+09,8.999999E+09,8.999999E+09]];
    LOCAL CONST Robtarget Tr_meulage_motif_1_274 := [[-37.6268203125,79.0580546875,35.2818515625],[0.363951430919515,-0.363241574410581,0.605870778174484,-0.607054787235555],[0,0,0,0],[8.999999E+09,8.999999E+09,8.999999E+09,8.999999E+09,8.999999E+09,8.999999E+09]];
    LOCAL CONST Robtarget Tr_meulage_motif_1_275 := [[-37.1551796875,79.93984375,35.281875],[0.363951430919515,-0.363241574410581,0.605870778174484,-0.607054787235555],[0,0,0,0],[8.999999E+09,8.999999E+09,8.999999E+09,8.999999E+09,8.999999E+09,8.999999E+09]];
    LOCAL CONST Robtarget Tr_meulage_motif_1_276 := [[-36.68354296875,80.821640625,35.28190234375],[0.363951430919515,-0.363241574410581,0.605870778174484,-0.607054787235555],[0,0,0,0],[8.999999E+09,8.999999E+09,8.999999E+09,8.999999E+09,8.999999E+09,8.999999E+09]];
    LOCAL CONST Robtarget Tr_meulage_motif_1_277 := [[-36.21190625,81.7034296875,35.28192578125],[0.363951430919515,-0.363241574410581,0.605870778174484,-0.607054787235555],[0,0,0,0],[8.999999E+09,8.999999E+09,8.999999E+09,8.999999E+09,8.999999E+09,8.999999E+09]];
    LOCAL CONST Robtarget Tr_meulage_motif_1_278 := [[-35.74026953125,82.5852265625,35.281953125],[0.363951430919515,-0.363241574410581,0.605870778174484,-0.607054787235555],[0,0,0,0],[8.999999E+09,8.999999E+09,8.999999E+09,8.999999E+09,8.999999E+09,8.999999E+09]];
    LOCAL CONST Robtarget Tr_meulage_motif_1_279 := [[-35.26862890625,83.467015625,35.2819765625],[0.363951430919515,-0.363241574410581,0.605870778174484,-0.607054787235555],[0,0,0,0],[8.999999E+09,8.999999E+09,8.999999E+09,8.999999E+09,8.999999E+09,8.999999E+09]];
    LOCAL CONST Robtarget Tr_meulage_motif_1_280 := [[-34.7969921875,84.3488046875,35.282],[0.363951430919515,-0.363241574410581,0.605870778174484,-0.607054787235555],[0,0,0,0],[8.999999E+09,8.999999E+09,8.999999E+09,8.999999E+09,8.999999E+09,8.999999E+09]];
    LOCAL CONST Robtarget Tr_meulage_motif_1_281 := [[-34.32535546875,85.2306015625,35.28202734375],[0.363951430919515,-0.363241574410581,0.605870778174484,-0.607054787235555],[0,0,0,0],[8.999999E+09,8.999999E+09,8.999999E+09,8.999999E+09,8.999999E+09,8.999999E+09]];
    LOCAL CONST Robtarget Tr_meulage_motif_1_282 := [[-33.85371875,86.112390625,35.28205078125],[0.363951430919515,-0.363241574410581,0.605870778174484,-0.607054787235555],[0,0,0,0],[8.999999E+09,8.999999E+09,8.999999E+09,8.999999E+09,8.999999E+09,8.999999E+09]];
    LOCAL CONST Robtarget Tr_meulage_motif_1_283 := [[-33.382078125,86.9941875,35.282078125],[0.363951430919515,-0.363241574410581,0.605870778174484,-0.607054787235555],[0,0,0,0],[8.999999E+09,8.999999E+09,8.999999E+09,8.999999E+09,8.999999E+09,8.999999E+09]];
    LOCAL CONST Robtarget Tr_meulage_motif_1_284 := [[-32.91044140625,87.8759765625,35.2821015625],[0.363951430919515,-0.363241574410581,0.605870778174484,-0.607054787235555],[0,0,0,0],[8.999999E+09,8.999999E+09,8.999999E+09,8.999999E+09,8.999999E+09,8.999999E+09]];
    LOCAL CONST Robtarget Tr_meulage_motif_1_285 := [[-32.4388046875,88.7577734375,35.28212890625],[0.363951430919515,-0.363241574410581,0.605870778174484,-0.607054787235555],[0,0,0,0],[8.999999E+09,8.999999E+09,8.999999E+09,8.999999E+09,8.999999E+09,8.999999E+09]];
    LOCAL CONST Robtarget Tr_meulage_motif_1_286 := [[-31.967166015625,89.6395625,35.28215234375],[0.363951430919515,-0.363241574410581,0.605870778174484,-0.607054787235555],[0,0,0,0],[8.999999E+09,8.999999E+09,8.999999E+09,8.999999E+09,8.999999E+09,8.999999E+09]];
    LOCAL CONST Robtarget Tr_meulage_motif_1_287 := [[-31.495529296875,90.5213515625,35.28217578125],[0.363951430919515,-0.363241574410581,0.605870778174484,-0.607054787235555],[0,0,0,0],[8.999999E+09,8.999999E+09,8.999999E+09,8.999999E+09,8.999999E+09,8.999999E+09]];
    LOCAL CONST Robtarget Tr_meulage_motif_1_288 := [[-31.023890625,91.4031484375,35.282203125],[0.363951430919515,-0.363241574410581,0.605870778174484,-0.607054787235555],[0,0,0,0],[8.999999E+09,8.999999E+09,8.999999E+09,8.999999E+09,8.999999E+09,8.999999E+09]];
    LOCAL CONST Robtarget Tr_meulage_motif_1_289 := [[-30.55225390625,92.2849375,35.2822265625],[0.363951430919515,-0.363241574410581,0.605870778174484,-0.607054787235555],[0,0,0,0],[8.999999E+09,8.999999E+09,8.999999E+09,8.999999E+09,8.999999E+09,8.999999E+09]];
    LOCAL CONST Robtarget Tr_meulage_motif_1_290 := [[-30.080615234375,93.166734375,35.28225390625],[0.363951430919515,-0.363241574410581,0.605870778174484,-0.607054787235555],[0,0,0,0],[8.999999E+09,8.999999E+09,8.999999E+09,8.999999E+09,8.999999E+09,8.999999E+09]];
    LOCAL CONST Robtarget Tr_meulage_motif_1_291 := [[-29.608978515625,94.0485234375,35.28227734375],[0.363951430919515,-0.363241574410581,0.605870778174484,-0.607054787235555],[0,0,0,0],[8.999999E+09,8.999999E+09,8.999999E+09,8.999999E+09,8.999999E+09,8.999999E+09]];
    LOCAL CONST Robtarget Tr_meulage_motif_1_292 := [[-29.13733984375,94.9303203125,35.2823046875],[0.363951430919515,-0.363241574410581,0.605870778174484,-0.607054787235555],[0,0,0,0],[8.999999E+09,8.999999E+09,8.999999E+09,8.999999E+09,8.999999E+09,8.999999E+09]];
    LOCAL CONST Robtarget Tr_meulage_motif_1_293 := [[-28.665703125,95.812109375,35.282328125],[0.363951430919515,-0.363241574410581,0.605870778174484,-0.607054787235555],[0,0,0,0],[8.999999E+09,8.999999E+09,8.999999E+09,8.999999E+09,8.999999E+09,8.999999E+09]];
    LOCAL CONST Robtarget Tr_meulage_motif_1_294 := [[-28.194064453125,96.6938984375,35.2823515625],[0.363951430919515,-0.363241574410581,0.605870778174484,-0.607054787235555],[0,0,0,0],[8.999999E+09,8.999999E+09,8.999999E+09,8.999999E+09,8.999999E+09,8.999999E+09]];

